// TwinCAT 3 PLC project PLC
// ProgramVersion: 3.1.4026.27
// libraries:
//   Tc2_MC2, * (Beckhoff Automation GmbH)
//   Tc2_MC2_Camming, * (Beckhoff Automation GmbH)
//   Tc2_Standard, * (Beckhoff Automation GmbH)
//   Tc2_System, * (Beckhoff Automation GmbH)
// project tree:
//   / PlcTask.TcTTO
//   DUTs/ E_Example.TcDUT, E_State.TcDUT, E_SegmentKind.TcDUT, ST_CamSegment.TcDUT, ST_CamSwitch.TcDUT
//   POUs/ F_CamPoint.TcPOU, FB_XtsBallCamBuilder.TcPOU, FB_XtsCamStitcher.TcPOU, MAIN.TcPOU, PRG_Example1.TcPOU, PRG_Example2.TcPOU, PRG_Example3.TcPOU, PRG_Example4.TcPOU, PRG_Example5.TcPOU
//   GVLs/ GVL_Axes.TcGVL
// real-time tasks:
//   TASK XTS Task 1: cycle T#250us, priority 1, ADS port 350
//   TASK XTS AUX Task 1: cycle T#250us, priority 2, ADS port 351
//   TASK PlcTask: cycle T#10ms, priority 20, ADS port 352
// motion (NC):
//   TASK NC-Task 1: cycle T#2ms, priority 4, ADS port 501
//   TASK NC-Task 1 SVB: cycle T#10ms, priority 8, ADS port 511
//   AXIS Mover Axis 1 (id 1)
//     Dynamic: AccelerationMaximum=80000, DecelerationMaximum=80000, Acceleration=20000, Deceleration=20000, Jerk=200000
//     Velo: Maximum=4000
//     PositionAreaControl: Enable=false
//     TargetPosControl: Enable=false
//     OtherSettings: AllowMotionCmdToSlave=true, AllowMotionCmdToExtSetGenAxis=true
//     encoder EncType=28
//       EncPara: ModuloFactor=1500, ToleranceWndModuloStart=0.2, MaxCount=#xffffffff
//     drive DrvType=22
//       DrvPara: MaxCount=#xffffffff, DriveControlDWord=#x00000100
//         Analog: VeloReferenz=4200, TorqueSetpointScale=10
//         TimeComp: TaskDelayCycles=1
//     controller CtrType=1
//       CtrPara: PriorControlFactor=1
//         PosDiffControl: Range=10
//         Observer: BandWidth=20
//   AXIS Mover Axis 2 (id 2)
//     Dynamic: AccelerationMaximum=80000, DecelerationMaximum=80000, Acceleration=20000, Deceleration=20000, Jerk=200000
//     Velo: Maximum=4000
//     PositionAreaControl: Enable=false
//     TargetPosControl: Enable=false
//     OtherSettings: AllowMotionCmdToSlave=true, AllowMotionCmdToExtSetGenAxis=true
//     encoder EncType=28
//       EncPara: ModuloFactor=1500, ToleranceWndModuloStart=0.2, MaxCount=#xffffffff
//     drive DrvType=22
//       DrvPara: MaxCount=#xffffffff, DriveControlDWord=#x00000100
//         Analog: VeloReferenz=4200, TorqueSetpointScale=10
//         TimeComp: TaskDelayCycles=1
//     controller CtrType=1
//       CtrPara: PriorControlFactor=1
//         PosDiffControl: Range=10
//         Observer: BandWidth=20
//   AXIS VirtualMaster (id 3)
//     General: UnitFlags=#x00000004
//     OtherSettings: AllowMotionCmdToSlave=true
//     encoder EncType=1
//       EncPara: ModuloFactor=2147.36
//     drive DrvType=5
//       Analog: TorqueSetpointScale=10, ScaleFactorActTorque=0.1
//       TimeComp: TaskDelayCycles=1
//     controller CtrType=1
//       CtrPara: PriorControlFactor=1
//         Observer: BandWidth=20
// I/O:
//   DEVICE Device 1 (disabled), AmsNetId 192.168.1.110.2.1
//     Term 0 (AT2001-0250) [AT2001-0250 Motor module with feed 250 mm, 48V]
//       Term 1 (AT2001-5250) [AT2001-5250 Sensor line with feed]
//     Term 2 (AT2050-0500) [AT2050-0500 Motor module, 90° clothoid, EtherCAT In, 48V]
//       Term 3 (AT2050-5500) [AT2050-5500 Sensor line 90° clothoid, EtherCAT In]
//     Term 4 (AT2050-0501) [AT2050-0501 Motor module, 90° clothoid, EtherCAT Out, 48V]
//       Term 5 (AT2050-5501) [AT2050-5501 Sensor line 90° clothoid, EtherCAT Out]
//     Term 6 (AT2000-0250) [AT2000-0250 Motor module 250 mm, 48V]
//       Term 7 (AT2000-5250) [AT2000-5250 Sensor line]
//     Term 8 (AT2050-0500) [AT2050-0500 Motor module, 90° clothoid, EtherCAT In, 48V]
//       Term 9 (AT2050-5500) [AT2050-5500 Sensor line 90° clothoid, EtherCAT In]
//     Term 10 (AT2050-0501) [AT2050-0501 Motor module, 90° clothoid, EtherCAT Out, 48V]
//       Term 11 (AT2050-5501) [AT2050-5501 Sensor line 90° clothoid, EtherCAT Out]
// variable links:
//   (this object) <-> TcCOM Objects/XTS ProcessingUnit 1/Part 1/Module 1
//     Term 0 (AT2001-0250)/CC Inputs/Current actual value Ch.1 <-> Data Pointer/CurrentActualValues[0]
//     Term 0 (AT2001-0250)/CC Inputs/Current actual value Ch.10 <-> Data Pointer/CurrentActualValues[9]
//     Term 0 (AT2001-0250)/CC Inputs/Current actual value Ch.11 <-> Data Pointer/CurrentActualValues[10]
//     Term 0 (AT2001-0250)/CC Inputs/Current actual value Ch.12 <-> Data Pointer/CurrentActualValues[11]
//     Term 0 (AT2001-0250)/CC Inputs/Current actual value Ch.13 <-> Data Pointer/CurrentActualValues[12]
//     Term 0 (AT2001-0250)/CC Inputs/Current actual value Ch.14 <-> Data Pointer/CurrentActualValues[13]
//     Term 0 (AT2001-0250)/CC Inputs/Current actual value Ch.15 <-> Data Pointer/CurrentActualValues[14]
//     Term 0 (AT2001-0250)/CC Inputs/Current actual value Ch.2 <-> Data Pointer/CurrentActualValues[1]
//     Term 0 (AT2001-0250)/CC Inputs/Current actual value Ch.3 <-> Data Pointer/CurrentActualValues[2]
//     Term 0 (AT2001-0250)/CC Inputs/Current actual value Ch.4 <-> Data Pointer/CurrentActualValues[3]
//     Term 0 (AT2001-0250)/CC Inputs/Current actual value Ch.5 <-> Data Pointer/CurrentActualValues[4]
//     Term 0 (AT2001-0250)/CC Inputs/Current actual value Ch.6 <-> Data Pointer/CurrentActualValues[5]
//     Term 0 (AT2001-0250)/CC Inputs/Current actual value Ch.7 <-> Data Pointer/CurrentActualValues[6]
//     Term 0 (AT2001-0250)/CC Inputs/Current actual value Ch.8 <-> Data Pointer/CurrentActualValues[7]
//     Term 0 (AT2001-0250)/CC Inputs/Current actual value Ch.9 <-> Data Pointer/CurrentActualValues[8]
//     Term 0 (AT2001-0250)/CC Inputs/Status <-> Data Pointer/Status
//     Term 0 (AT2001-0250)/CC Outputs/Control <-> Data Pointer/Control
//     Term 0 (AT2001-0250)/CC Outputs/Current setpoint value Ch.1 <-> Data Pointer/CurrentSetpointValues[0]
//     Term 0 (AT2001-0250)/CC Outputs/Current setpoint value Ch.10 <-> Data Pointer/CurrentSetpointValues[9]
//     Term 0 (AT2001-0250)/CC Outputs/Current setpoint value Ch.11 <-> Data Pointer/CurrentSetpointValues[10]
//     Term 0 (AT2001-0250)/CC Outputs/Current setpoint value Ch.12 <-> Data Pointer/CurrentSetpointValues[11]
//     Term 0 (AT2001-0250)/CC Outputs/Current setpoint value Ch.13 <-> Data Pointer/CurrentSetpointValues[12]
//     Term 0 (AT2001-0250)/CC Outputs/Current setpoint value Ch.14 <-> Data Pointer/CurrentSetpointValues[13]
//     Term 0 (AT2001-0250)/CC Outputs/Current setpoint value Ch.15 <-> Data Pointer/CurrentSetpointValues[14]
//     Term 0 (AT2001-0250)/CC Outputs/Current setpoint value Ch.2 <-> Data Pointer/CurrentSetpointValues[1]
//     Term 0 (AT2001-0250)/CC Outputs/Current setpoint value Ch.3 <-> Data Pointer/CurrentSetpointValues[2]
//     Term 0 (AT2001-0250)/CC Outputs/Current setpoint value Ch.4 <-> Data Pointer/CurrentSetpointValues[3]
//     Term 0 (AT2001-0250)/CC Outputs/Current setpoint value Ch.5 <-> Data Pointer/CurrentSetpointValues[4]
//     Term 0 (AT2001-0250)/CC Outputs/Current setpoint value Ch.6 <-> Data Pointer/CurrentSetpointValues[5]
//     Term 0 (AT2001-0250)/CC Outputs/Current setpoint value Ch.7 <-> Data Pointer/CurrentSetpointValues[6]
//     Term 0 (AT2001-0250)/CC Outputs/Current setpoint value Ch.8 <-> Data Pointer/CurrentSetpointValues[7]
//     Term 0 (AT2001-0250)/CC Outputs/Current setpoint value Ch.9 <-> Data Pointer/CurrentSetpointValues[8]
//     Term 0 (AT2001-0250)/Term 1 (AT2001-5250)/FB Inputs/Value Channel 01 <-> Data Pointer/RawPositionValues[0]
//     Term 0 (AT2001-0250)/Term 1 (AT2001-5250)/FB Inputs/Value Channel 02 <-> Data Pointer/RawPositionValues[1]
//     Term 0 (AT2001-0250)/Term 1 (AT2001-5250)/FB Inputs/Value Channel 03 <-> Data Pointer/RawPositionValues[2]
//     Term 0 (AT2001-0250)/Term 1 (AT2001-5250)/FB Inputs/Value Channel 04 <-> Data Pointer/RawPositionValues[3]
//     Term 0 (AT2001-0250)/Term 1 (AT2001-5250)/FB Inputs/Value Channel 05 <-> Data Pointer/RawPositionValues[4]
//     Term 0 (AT2001-0250)/Term 1 (AT2001-5250)/FB Inputs/Value Channel 06 <-> Data Pointer/RawPositionValues[5]
//     Term 0 (AT2001-0250)/Term 1 (AT2001-5250)/FB Inputs/Value Channel 07 <-> Data Pointer/RawPositionValues[6]
//     Term 0 (AT2001-0250)/Term 1 (AT2001-5250)/FB Inputs/Value Channel 08 <-> Data Pointer/RawPositionValues[7]
//     Term 0 (AT2001-0250)/Term 1 (AT2001-5250)/FB Inputs/Value Channel 09 <-> Data Pointer/RawPositionValues[8]
//     Term 0 (AT2001-0250)/Term 1 (AT2001-5250)/FB Inputs/Value Channel 10 <-> Data Pointer/RawPositionValues[9]
//     Term 0 (AT2001-0250)/Term 1 (AT2001-5250)/FB Inputs/Value Channel 11 <-> Data Pointer/RawPositionValues[10]
//     Term 0 (AT2001-0250)/Term 1 (AT2001-5250)/FB Inputs/Value Channel 12 <-> Data Pointer/RawPositionValues[11]
//     Term 0 (AT2001-0250)/Term 1 (AT2001-5250)/FB Inputs/Value Channel 13 <-> Data Pointer/RawPositionValues[12]
//     Term 0 (AT2001-0250)/Term 1 (AT2001-5250)/FB Inputs/Value Channel 14 <-> Data Pointer/RawPositionValues[13]
//     Term 0 (AT2001-0250)/Term 1 (AT2001-5250)/FB Inputs/Value Channel 15 <-> Data Pointer/RawPositionValues[14]
//     Term 0 (AT2001-0250)/Term 1 (AT2001-5250)/FB Inputs/Value Channel 16 <-> Data Pointer/RawPositionValues[15]
//     Term 0 (AT2001-0250)/Term 1 (AT2001-5250)/FB Inputs/Value Channel 17 <-> Data Pointer/RawPositionValues[16]
//     Term 0 (AT2001-0250)/Term 1 (AT2001-5250)/FB Inputs/Value Channel 18 <-> Data Pointer/RawPositionValues[17]
//     Term 0 (AT2001-0250)/Term 1 (AT2001-5250)/FB Inputs/Value Channel 19 <-> Data Pointer/RawPositionValues[18]
//     Term 0 (AT2001-0250)/Term 1 (AT2001-5250)/FB Inputs/Value Channel 20 <-> Data Pointer/RawPositionValues[19]
//     Term 0 (AT2001-0250)/Term 1 (AT2001-5250)/FB Inputs/Value Channel 21 <-> Data Pointer/RawPositionValues[20]
//     Term 0 (AT2001-0250)/Term 1 (AT2001-5250)/FB Inputs/Value Channel 22 <-> Data Pointer/RawPositionValues[21]
//     Term 0 (AT2001-0250)/Term 1 (AT2001-5250)/FB Inputs/Value Channel 23 <-> Data Pointer/RawPositionValues[22]
//     Term 0 (AT2001-0250)/Term 1 (AT2001-5250)/FB Inputs/Value Channel 24 <-> Data Pointer/RawPositionValues[23]
//     Term 0 (AT2001-0250)/Term 1 (AT2001-5250)/FB Inputs/Value Channel 25 <-> Data Pointer/RawPositionValues[24]
//     Term 0 (AT2001-0250)/Term 1 (AT2001-5250)/FB Inputs/Value Channel 26 <-> Data Pointer/RawPositionValues[25]
//     Term 0 (AT2001-0250)/Term 1 (AT2001-5250)/FB Inputs/Value Channel 27 <-> Data Pointer/RawPositionValues[26]
//     Term 0 (AT2001-0250)/Term 1 (AT2001-5250)/FB Inputs/Value Channel 28 <-> Data Pointer/RawPositionValues[27]
//     Term 0 (AT2001-0250)/Term 1 (AT2001-5250)/FB Inputs/Value Channel 29 <-> Data Pointer/RawPositionValues[28]
//     Term 0 (AT2001-0250)/Term 1 (AT2001-5250)/FB Inputs/Value Channel 30 <-> Data Pointer/RawPositionValues[29]
//     Term 0 (AT2001-0250)/Term 1 (AT2001-5250)/FB Inputs/Value Channel 31 <-> Data Pointer/RawPositionValues[30]
//     Term 0 (AT2001-0250)/Term 1 (AT2001-5250)/FB Inputs/Value Channel 32 <-> Data Pointer/RawPositionValues[31]
//   (this object) <-> TcCOM Objects/XTS ProcessingUnit 1/Part 1/Module 2
//     Term 2 (AT2050-0500)/CC Inputs/Current actual value Ch.1 <-> Data Pointer/CurrentActualValues[0]
//     Term 2 (AT2050-0500)/CC Inputs/Current actual value Ch.10 <-> Data Pointer/CurrentActualValues[9]
//     Term 2 (AT2050-0500)/CC Inputs/Current actual value Ch.11 <-> Data Pointer/CurrentActualValues[10]
//     Term 2 (AT2050-0500)/CC Inputs/Current actual value Ch.12 <-> Data Pointer/CurrentActualValues[11]
//     Term 2 (AT2050-0500)/CC Inputs/Current actual value Ch.13 <-> Data Pointer/CurrentActualValues[12]
//     Term 2 (AT2050-0500)/CC Inputs/Current actual value Ch.14 <-> Data Pointer/CurrentActualValues[13]
//     Term 2 (AT2050-0500)/CC Inputs/Current actual value Ch.15 <-> Data Pointer/CurrentActualValues[14]
//     Term 2 (AT2050-0500)/CC Inputs/Current actual value Ch.2 <-> Data Pointer/CurrentActualValues[1]
//     Term 2 (AT2050-0500)/CC Inputs/Current actual value Ch.3 <-> Data Pointer/CurrentActualValues[2]
//     Term 2 (AT2050-0500)/CC Inputs/Current actual value Ch.4 <-> Data Pointer/CurrentActualValues[3]
//     Term 2 (AT2050-0500)/CC Inputs/Current actual value Ch.5 <-> Data Pointer/CurrentActualValues[4]
//     Term 2 (AT2050-0500)/CC Inputs/Current actual value Ch.6 <-> Data Pointer/CurrentActualValues[5]
//     Term 2 (AT2050-0500)/CC Inputs/Current actual value Ch.7 <-> Data Pointer/CurrentActualValues[6]
//     Term 2 (AT2050-0500)/CC Inputs/Current actual value Ch.8 <-> Data Pointer/CurrentActualValues[7]
//     Term 2 (AT2050-0500)/CC Inputs/Current actual value Ch.9 <-> Data Pointer/CurrentActualValues[8]
//     Term 2 (AT2050-0500)/CC Inputs/Status <-> Data Pointer/Status
//     Term 2 (AT2050-0500)/CC Outputs/Control <-> Data Pointer/Control
//     Term 2 (AT2050-0500)/CC Outputs/Current setpoint value Ch.1 <-> Data Pointer/CurrentSetpointValues[0]
//     Term 2 (AT2050-0500)/CC Outputs/Current setpoint value Ch.10 <-> Data Pointer/CurrentSetpointValues[9]
//     Term 2 (AT2050-0500)/CC Outputs/Current setpoint value Ch.11 <-> Data Pointer/CurrentSetpointValues[10]
//     Term 2 (AT2050-0500)/CC Outputs/Current setpoint value Ch.12 <-> Data Pointer/CurrentSetpointValues[11]
//     Term 2 (AT2050-0500)/CC Outputs/Current setpoint value Ch.13 <-> Data Pointer/CurrentSetpointValues[12]
//     Term 2 (AT2050-0500)/CC Outputs/Current setpoint value Ch.14 <-> Data Pointer/CurrentSetpointValues[13]
//     Term 2 (AT2050-0500)/CC Outputs/Current setpoint value Ch.15 <-> Data Pointer/CurrentSetpointValues[14]
//     Term 2 (AT2050-0500)/CC Outputs/Current setpoint value Ch.2 <-> Data Pointer/CurrentSetpointValues[1]
//     Term 2 (AT2050-0500)/CC Outputs/Current setpoint value Ch.3 <-> Data Pointer/CurrentSetpointValues[2]
//     Term 2 (AT2050-0500)/CC Outputs/Current setpoint value Ch.4 <-> Data Pointer/CurrentSetpointValues[3]
//     Term 2 (AT2050-0500)/CC Outputs/Current setpoint value Ch.5 <-> Data Pointer/CurrentSetpointValues[4]
//     Term 2 (AT2050-0500)/CC Outputs/Current setpoint value Ch.6 <-> Data Pointer/CurrentSetpointValues[5]
//     Term 2 (AT2050-0500)/CC Outputs/Current setpoint value Ch.7 <-> Data Pointer/CurrentSetpointValues[6]
//     Term 2 (AT2050-0500)/CC Outputs/Current setpoint value Ch.8 <-> Data Pointer/CurrentSetpointValues[7]
//     Term 2 (AT2050-0500)/CC Outputs/Current setpoint value Ch.9 <-> Data Pointer/CurrentSetpointValues[8]
//     Term 2 (AT2050-0500)/Term 3 (AT2050-5500)/FB Inputs/Value Channel 01 <-> Data Pointer/RawPositionValues[0]
//     Term 2 (AT2050-0500)/Term 3 (AT2050-5500)/FB Inputs/Value Channel 02 <-> Data Pointer/RawPositionValues[1]
//     Term 2 (AT2050-0500)/Term 3 (AT2050-5500)/FB Inputs/Value Channel 03 <-> Data Pointer/RawPositionValues[2]
//     Term 2 (AT2050-0500)/Term 3 (AT2050-5500)/FB Inputs/Value Channel 04 <-> Data Pointer/RawPositionValues[3]
//     Term 2 (AT2050-0500)/Term 3 (AT2050-5500)/FB Inputs/Value Channel 05 <-> Data Pointer/RawPositionValues[4]
//     Term 2 (AT2050-0500)/Term 3 (AT2050-5500)/FB Inputs/Value Channel 06 <-> Data Pointer/RawPositionValues[5]
//     Term 2 (AT2050-0500)/Term 3 (AT2050-5500)/FB Inputs/Value Channel 07 <-> Data Pointer/RawPositionValues[6]
//     Term 2 (AT2050-0500)/Term 3 (AT2050-5500)/FB Inputs/Value Channel 08 <-> Data Pointer/RawPositionValues[7]
//     Term 2 (AT2050-0500)/Term 3 (AT2050-5500)/FB Inputs/Value Channel 09 <-> Data Pointer/RawPositionValues[8]
//     Term 2 (AT2050-0500)/Term 3 (AT2050-5500)/FB Inputs/Value Channel 10 <-> Data Pointer/RawPositionValues[9]
//     Term 2 (AT2050-0500)/Term 3 (AT2050-5500)/FB Inputs/Value Channel 11 <-> Data Pointer/RawPositionValues[10]
//     Term 2 (AT2050-0500)/Term 3 (AT2050-5500)/FB Inputs/Value Channel 12 <-> Data Pointer/RawPositionValues[11]
//     Term 2 (AT2050-0500)/Term 3 (AT2050-5500)/FB Inputs/Value Channel 13 <-> Data Pointer/RawPositionValues[12]
//     Term 2 (AT2050-0500)/Term 3 (AT2050-5500)/FB Inputs/Value Channel 14 <-> Data Pointer/RawPositionValues[13]
//     Term 2 (AT2050-0500)/Term 3 (AT2050-5500)/FB Inputs/Value Channel 15 <-> Data Pointer/RawPositionValues[14]
//     Term 2 (AT2050-0500)/Term 3 (AT2050-5500)/FB Inputs/Value Channel 16 <-> Data Pointer/RawPositionValues[15]
//     Term 2 (AT2050-0500)/Term 3 (AT2050-5500)/FB Inputs/Value Channel 17 <-> Data Pointer/RawPositionValues[16]
//     Term 2 (AT2050-0500)/Term 3 (AT2050-5500)/FB Inputs/Value Channel 18 <-> Data Pointer/RawPositionValues[17]
//     Term 2 (AT2050-0500)/Term 3 (AT2050-5500)/FB Inputs/Value Channel 19 <-> Data Pointer/RawPositionValues[18]
//     Term 2 (AT2050-0500)/Term 3 (AT2050-5500)/FB Inputs/Value Channel 20 <-> Data Pointer/RawPositionValues[19]
//     Term 2 (AT2050-0500)/Term 3 (AT2050-5500)/FB Inputs/Value Channel 21 <-> Data Pointer/RawPositionValues[20]
//     Term 2 (AT2050-0500)/Term 3 (AT2050-5500)/FB Inputs/Value Channel 22 <-> Data Pointer/RawPositionValues[21]
//     Term 2 (AT2050-0500)/Term 3 (AT2050-5500)/FB Inputs/Value Channel 23 <-> Data Pointer/RawPositionValues[22]
//     Term 2 (AT2050-0500)/Term 3 (AT2050-5500)/FB Inputs/Value Channel 24 <-> Data Pointer/RawPositionValues[23]
//     Term 2 (AT2050-0500)/Term 3 (AT2050-5500)/FB Inputs/Value Channel 25 <-> Data Pointer/RawPositionValues[24]
//     Term 2 (AT2050-0500)/Term 3 (AT2050-5500)/FB Inputs/Value Channel 26 <-> Data Pointer/RawPositionValues[25]
//     Term 2 (AT2050-0500)/Term 3 (AT2050-5500)/FB Inputs/Value Channel 27 <-> Data Pointer/RawPositionValues[26]
//     Term 2 (AT2050-0500)/Term 3 (AT2050-5500)/FB Inputs/Value Channel 28 <-> Data Pointer/RawPositionValues[27]
//     Term 2 (AT2050-0500)/Term 3 (AT2050-5500)/FB Inputs/Value Channel 29 <-> Data Pointer/RawPositionValues[28]
//     Term 2 (AT2050-0500)/Term 3 (AT2050-5500)/FB Inputs/Value Channel 30 <-> Data Pointer/RawPositionValues[29]
//     Term 2 (AT2050-0500)/Term 3 (AT2050-5500)/FB Inputs/Value Channel 31 <-> Data Pointer/RawPositionValues[30]
//     Term 2 (AT2050-0500)/Term 3 (AT2050-5500)/FB Inputs/Value Channel 32 <-> Data Pointer/RawPositionValues[31]
//   (this object) <-> TcCOM Objects/XTS ProcessingUnit 1/Part 1/Module 3
//     Term 4 (AT2050-0501)/CC Inputs/Current actual value Ch.1 <-> Data Pointer/CurrentActualValues[0]
//     Term 4 (AT2050-0501)/CC Inputs/Current actual value Ch.10 <-> Data Pointer/CurrentActualValues[9]
//     Term 4 (AT2050-0501)/CC Inputs/Current actual value Ch.11 <-> Data Pointer/CurrentActualValues[10]
//     Term 4 (AT2050-0501)/CC Inputs/Current actual value Ch.12 <-> Data Pointer/CurrentActualValues[11]
//     Term 4 (AT2050-0501)/CC Inputs/Current actual value Ch.13 <-> Data Pointer/CurrentActualValues[12]
//     Term 4 (AT2050-0501)/CC Inputs/Current actual value Ch.14 <-> Data Pointer/CurrentActualValues[13]
//     Term 4 (AT2050-0501)/CC Inputs/Current actual value Ch.15 <-> Data Pointer/CurrentActualValues[14]
//     Term 4 (AT2050-0501)/CC Inputs/Current actual value Ch.2 <-> Data Pointer/CurrentActualValues[1]
//     Term 4 (AT2050-0501)/CC Inputs/Current actual value Ch.3 <-> Data Pointer/CurrentActualValues[2]
//     Term 4 (AT2050-0501)/CC Inputs/Current actual value Ch.4 <-> Data Pointer/CurrentActualValues[3]
//     Term 4 (AT2050-0501)/CC Inputs/Current actual value Ch.5 <-> Data Pointer/CurrentActualValues[4]
//     Term 4 (AT2050-0501)/CC Inputs/Current actual value Ch.6 <-> Data Pointer/CurrentActualValues[5]
//     Term 4 (AT2050-0501)/CC Inputs/Current actual value Ch.7 <-> Data Pointer/CurrentActualValues[6]
//     Term 4 (AT2050-0501)/CC Inputs/Current actual value Ch.8 <-> Data Pointer/CurrentActualValues[7]
//     Term 4 (AT2050-0501)/CC Inputs/Current actual value Ch.9 <-> Data Pointer/CurrentActualValues[8]
//     Term 4 (AT2050-0501)/CC Inputs/Status <-> Data Pointer/Status
//     Term 4 (AT2050-0501)/CC Outputs/Control <-> Data Pointer/Control
//     Term 4 (AT2050-0501)/CC Outputs/Current setpoint value Ch.1 <-> Data Pointer/CurrentSetpointValues[0]
//     Term 4 (AT2050-0501)/CC Outputs/Current setpoint value Ch.10 <-> Data Pointer/CurrentSetpointValues[9]
//     Term 4 (AT2050-0501)/CC Outputs/Current setpoint value Ch.11 <-> Data Pointer/CurrentSetpointValues[10]
//     Term 4 (AT2050-0501)/CC Outputs/Current setpoint value Ch.12 <-> Data Pointer/CurrentSetpointValues[11]
//     Term 4 (AT2050-0501)/CC Outputs/Current setpoint value Ch.13 <-> Data Pointer/CurrentSetpointValues[12]
//     Term 4 (AT2050-0501)/CC Outputs/Current setpoint value Ch.14 <-> Data Pointer/CurrentSetpointValues[13]
//     Term 4 (AT2050-0501)/CC Outputs/Current setpoint value Ch.15 <-> Data Pointer/CurrentSetpointValues[14]
//     Term 4 (AT2050-0501)/CC Outputs/Current setpoint value Ch.2 <-> Data Pointer/CurrentSetpointValues[1]
//     Term 4 (AT2050-0501)/CC Outputs/Current setpoint value Ch.3 <-> Data Pointer/CurrentSetpointValues[2]
//     Term 4 (AT2050-0501)/CC Outputs/Current setpoint value Ch.4 <-> Data Pointer/CurrentSetpointValues[3]
//     Term 4 (AT2050-0501)/CC Outputs/Current setpoint value Ch.5 <-> Data Pointer/CurrentSetpointValues[4]
//     Term 4 (AT2050-0501)/CC Outputs/Current setpoint value Ch.6 <-> Data Pointer/CurrentSetpointValues[5]
//     Term 4 (AT2050-0501)/CC Outputs/Current setpoint value Ch.7 <-> Data Pointer/CurrentSetpointValues[6]
//     Term 4 (AT2050-0501)/CC Outputs/Current setpoint value Ch.8 <-> Data Pointer/CurrentSetpointValues[7]
//     Term 4 (AT2050-0501)/CC Outputs/Current setpoint value Ch.9 <-> Data Pointer/CurrentSetpointValues[8]
//     Term 4 (AT2050-0501)/Term 5 (AT2050-5501)/FB Inputs/Value Channel 01 <-> Data Pointer/RawPositionValues[0]
//     Term 4 (AT2050-0501)/Term 5 (AT2050-5501)/FB Inputs/Value Channel 02 <-> Data Pointer/RawPositionValues[1]
//     Term 4 (AT2050-0501)/Term 5 (AT2050-5501)/FB Inputs/Value Channel 03 <-> Data Pointer/RawPositionValues[2]
//     Term 4 (AT2050-0501)/Term 5 (AT2050-5501)/FB Inputs/Value Channel 04 <-> Data Pointer/RawPositionValues[3]
//     Term 4 (AT2050-0501)/Term 5 (AT2050-5501)/FB Inputs/Value Channel 05 <-> Data Pointer/RawPositionValues[4]
//     Term 4 (AT2050-0501)/Term 5 (AT2050-5501)/FB Inputs/Value Channel 06 <-> Data Pointer/RawPositionValues[5]
//     Term 4 (AT2050-0501)/Term 5 (AT2050-5501)/FB Inputs/Value Channel 07 <-> Data Pointer/RawPositionValues[6]
//     Term 4 (AT2050-0501)/Term 5 (AT2050-5501)/FB Inputs/Value Channel 08 <-> Data Pointer/RawPositionValues[7]
//     Term 4 (AT2050-0501)/Term 5 (AT2050-5501)/FB Inputs/Value Channel 09 <-> Data Pointer/RawPositionValues[8]
//     Term 4 (AT2050-0501)/Term 5 (AT2050-5501)/FB Inputs/Value Channel 10 <-> Data Pointer/RawPositionValues[9]
//     Term 4 (AT2050-0501)/Term 5 (AT2050-5501)/FB Inputs/Value Channel 11 <-> Data Pointer/RawPositionValues[10]
//     Term 4 (AT2050-0501)/Term 5 (AT2050-5501)/FB Inputs/Value Channel 12 <-> Data Pointer/RawPositionValues[11]
//     Term 4 (AT2050-0501)/Term 5 (AT2050-5501)/FB Inputs/Value Channel 13 <-> Data Pointer/RawPositionValues[12]
//     Term 4 (AT2050-0501)/Term 5 (AT2050-5501)/FB Inputs/Value Channel 14 <-> Data Pointer/RawPositionValues[13]
//     Term 4 (AT2050-0501)/Term 5 (AT2050-5501)/FB Inputs/Value Channel 15 <-> Data Pointer/RawPositionValues[14]
//     Term 4 (AT2050-0501)/Term 5 (AT2050-5501)/FB Inputs/Value Channel 16 <-> Data Pointer/RawPositionValues[15]
//     Term 4 (AT2050-0501)/Term 5 (AT2050-5501)/FB Inputs/Value Channel 17 <-> Data Pointer/RawPositionValues[16]
//     Term 4 (AT2050-0501)/Term 5 (AT2050-5501)/FB Inputs/Value Channel 18 <-> Data Pointer/RawPositionValues[17]
//     Term 4 (AT2050-0501)/Term 5 (AT2050-5501)/FB Inputs/Value Channel 19 <-> Data Pointer/RawPositionValues[18]
//     Term 4 (AT2050-0501)/Term 5 (AT2050-5501)/FB Inputs/Value Channel 20 <-> Data Pointer/RawPositionValues[19]
//     Term 4 (AT2050-0501)/Term 5 (AT2050-5501)/FB Inputs/Value Channel 21 <-> Data Pointer/RawPositionValues[20]
//     Term 4 (AT2050-0501)/Term 5 (AT2050-5501)/FB Inputs/Value Channel 22 <-> Data Pointer/RawPositionValues[21]
//     Term 4 (AT2050-0501)/Term 5 (AT2050-5501)/FB Inputs/Value Channel 23 <-> Data Pointer/RawPositionValues[22]
//     Term 4 (AT2050-0501)/Term 5 (AT2050-5501)/FB Inputs/Value Channel 24 <-> Data Pointer/RawPositionValues[23]
//     Term 4 (AT2050-0501)/Term 5 (AT2050-5501)/FB Inputs/Value Channel 25 <-> Data Pointer/RawPositionValues[24]
//     Term 4 (AT2050-0501)/Term 5 (AT2050-5501)/FB Inputs/Value Channel 26 <-> Data Pointer/RawPositionValues[25]
//     Term 4 (AT2050-0501)/Term 5 (AT2050-5501)/FB Inputs/Value Channel 27 <-> Data Pointer/RawPositionValues[26]
//     Term 4 (AT2050-0501)/Term 5 (AT2050-5501)/FB Inputs/Value Channel 28 <-> Data Pointer/RawPositionValues[27]
//     Term 4 (AT2050-0501)/Term 5 (AT2050-5501)/FB Inputs/Value Channel 29 <-> Data Pointer/RawPositionValues[28]
//     Term 4 (AT2050-0501)/Term 5 (AT2050-5501)/FB Inputs/Value Channel 30 <-> Data Pointer/RawPositionValues[29]
//     Term 4 (AT2050-0501)/Term 5 (AT2050-5501)/FB Inputs/Value Channel 31 <-> Data Pointer/RawPositionValues[30]
//     Term 4 (AT2050-0501)/Term 5 (AT2050-5501)/FB Inputs/Value Channel 32 <-> Data Pointer/RawPositionValues[31]
//   (this object) <-> TcCOM Objects/XTS ProcessingUnit 1/Part 1/Module 4
//     Term 6 (AT2000-0250)/CC Inputs/Current actual value Ch.1 <-> Data Pointer/CurrentActualValues[0]
//     Term 6 (AT2000-0250)/CC Inputs/Current actual value Ch.10 <-> Data Pointer/CurrentActualValues[9]
//     Term 6 (AT2000-0250)/CC Inputs/Current actual value Ch.11 <-> Data Pointer/CurrentActualValues[10]
//     Term 6 (AT2000-0250)/CC Inputs/Current actual value Ch.12 <-> Data Pointer/CurrentActualValues[11]
//     Term 6 (AT2000-0250)/CC Inputs/Current actual value Ch.13 <-> Data Pointer/CurrentActualValues[12]
//     Term 6 (AT2000-0250)/CC Inputs/Current actual value Ch.14 <-> Data Pointer/CurrentActualValues[13]
//     Term 6 (AT2000-0250)/CC Inputs/Current actual value Ch.15 <-> Data Pointer/CurrentActualValues[14]
//     Term 6 (AT2000-0250)/CC Inputs/Current actual value Ch.2 <-> Data Pointer/CurrentActualValues[1]
//     Term 6 (AT2000-0250)/CC Inputs/Current actual value Ch.3 <-> Data Pointer/CurrentActualValues[2]
//     Term 6 (AT2000-0250)/CC Inputs/Current actual value Ch.4 <-> Data Pointer/CurrentActualValues[3]
//     Term 6 (AT2000-0250)/CC Inputs/Current actual value Ch.5 <-> Data Pointer/CurrentActualValues[4]
//     Term 6 (AT2000-0250)/CC Inputs/Current actual value Ch.6 <-> Data Pointer/CurrentActualValues[5]
//     Term 6 (AT2000-0250)/CC Inputs/Current actual value Ch.7 <-> Data Pointer/CurrentActualValues[6]
//     Term 6 (AT2000-0250)/CC Inputs/Current actual value Ch.8 <-> Data Pointer/CurrentActualValues[7]
//     Term 6 (AT2000-0250)/CC Inputs/Current actual value Ch.9 <-> Data Pointer/CurrentActualValues[8]
//     Term 6 (AT2000-0250)/CC Inputs/Status <-> Data Pointer/Status
//     Term 6 (AT2000-0250)/CC Outputs/Control <-> Data Pointer/Control
//     Term 6 (AT2000-0250)/CC Outputs/Current setpoint value Ch.1 <-> Data Pointer/CurrentSetpointValues[0]
//     Term 6 (AT2000-0250)/CC Outputs/Current setpoint value Ch.10 <-> Data Pointer/CurrentSetpointValues[9]
//     Term 6 (AT2000-0250)/CC Outputs/Current setpoint value Ch.11 <-> Data Pointer/CurrentSetpointValues[10]
//     Term 6 (AT2000-0250)/CC Outputs/Current setpoint value Ch.12 <-> Data Pointer/CurrentSetpointValues[11]
//     Term 6 (AT2000-0250)/CC Outputs/Current setpoint value Ch.13 <-> Data Pointer/CurrentSetpointValues[12]
//     Term 6 (AT2000-0250)/CC Outputs/Current setpoint value Ch.14 <-> Data Pointer/CurrentSetpointValues[13]
//     Term 6 (AT2000-0250)/CC Outputs/Current setpoint value Ch.15 <-> Data Pointer/CurrentSetpointValues[14]
//     Term 6 (AT2000-0250)/CC Outputs/Current setpoint value Ch.2 <-> Data Pointer/CurrentSetpointValues[1]
//     Term 6 (AT2000-0250)/CC Outputs/Current setpoint value Ch.3 <-> Data Pointer/CurrentSetpointValues[2]
//     Term 6 (AT2000-0250)/CC Outputs/Current setpoint value Ch.4 <-> Data Pointer/CurrentSetpointValues[3]
//     Term 6 (AT2000-0250)/CC Outputs/Current setpoint value Ch.5 <-> Data Pointer/CurrentSetpointValues[4]
//     Term 6 (AT2000-0250)/CC Outputs/Current setpoint value Ch.6 <-> Data Pointer/CurrentSetpointValues[5]
//     Term 6 (AT2000-0250)/CC Outputs/Current setpoint value Ch.7 <-> Data Pointer/CurrentSetpointValues[6]
//     Term 6 (AT2000-0250)/CC Outputs/Current setpoint value Ch.8 <-> Data Pointer/CurrentSetpointValues[7]
//     Term 6 (AT2000-0250)/CC Outputs/Current setpoint value Ch.9 <-> Data Pointer/CurrentSetpointValues[8]
//     Term 6 (AT2000-0250)/Term 7 (AT2000-5250)/FB Inputs/Value Channel 01 <-> Data Pointer/RawPositionValues[0]
//     Term 6 (AT2000-0250)/Term 7 (AT2000-5250)/FB Inputs/Value Channel 02 <-> Data Pointer/RawPositionValues[1]
//     Term 6 (AT2000-0250)/Term 7 (AT2000-5250)/FB Inputs/Value Channel 03 <-> Data Pointer/RawPositionValues[2]
//     Term 6 (AT2000-0250)/Term 7 (AT2000-5250)/FB Inputs/Value Channel 04 <-> Data Pointer/RawPositionValues[3]
//     Term 6 (AT2000-0250)/Term 7 (AT2000-5250)/FB Inputs/Value Channel 05 <-> Data Pointer/RawPositionValues[4]
//     Term 6 (AT2000-0250)/Term 7 (AT2000-5250)/FB Inputs/Value Channel 06 <-> Data Pointer/RawPositionValues[5]
//     Term 6 (AT2000-0250)/Term 7 (AT2000-5250)/FB Inputs/Value Channel 07 <-> Data Pointer/RawPositionValues[6]
//     Term 6 (AT2000-0250)/Term 7 (AT2000-5250)/FB Inputs/Value Channel 08 <-> Data Pointer/RawPositionValues[7]
//     Term 6 (AT2000-0250)/Term 7 (AT2000-5250)/FB Inputs/Value Channel 09 <-> Data Pointer/RawPositionValues[8]
//     Term 6 (AT2000-0250)/Term 7 (AT2000-5250)/FB Inputs/Value Channel 10 <-> Data Pointer/RawPositionValues[9]
//     Term 6 (AT2000-0250)/Term 7 (AT2000-5250)/FB Inputs/Value Channel 11 <-> Data Pointer/RawPositionValues[10]
//     Term 6 (AT2000-0250)/Term 7 (AT2000-5250)/FB Inputs/Value Channel 12 <-> Data Pointer/RawPositionValues[11]
//     Term 6 (AT2000-0250)/Term 7 (AT2000-5250)/FB Inputs/Value Channel 13 <-> Data Pointer/RawPositionValues[12]
//     Term 6 (AT2000-0250)/Term 7 (AT2000-5250)/FB Inputs/Value Channel 14 <-> Data Pointer/RawPositionValues[13]
//     Term 6 (AT2000-0250)/Term 7 (AT2000-5250)/FB Inputs/Value Channel 15 <-> Data Pointer/RawPositionValues[14]
//     Term 6 (AT2000-0250)/Term 7 (AT2000-5250)/FB Inputs/Value Channel 16 <-> Data Pointer/RawPositionValues[15]
//     Term 6 (AT2000-0250)/Term 7 (AT2000-5250)/FB Inputs/Value Channel 17 <-> Data Pointer/RawPositionValues[16]
//     Term 6 (AT2000-0250)/Term 7 (AT2000-5250)/FB Inputs/Value Channel 18 <-> Data Pointer/RawPositionValues[17]
//     Term 6 (AT2000-0250)/Term 7 (AT2000-5250)/FB Inputs/Value Channel 19 <-> Data Pointer/RawPositionValues[18]
//     Term 6 (AT2000-0250)/Term 7 (AT2000-5250)/FB Inputs/Value Channel 20 <-> Data Pointer/RawPositionValues[19]
//     Term 6 (AT2000-0250)/Term 7 (AT2000-5250)/FB Inputs/Value Channel 21 <-> Data Pointer/RawPositionValues[20]
//     Term 6 (AT2000-0250)/Term 7 (AT2000-5250)/FB Inputs/Value Channel 22 <-> Data Pointer/RawPositionValues[21]
//     Term 6 (AT2000-0250)/Term 7 (AT2000-5250)/FB Inputs/Value Channel 23 <-> Data Pointer/RawPositionValues[22]
//     Term 6 (AT2000-0250)/Term 7 (AT2000-5250)/FB Inputs/Value Channel 24 <-> Data Pointer/RawPositionValues[23]
//     Term 6 (AT2000-0250)/Term 7 (AT2000-5250)/FB Inputs/Value Channel 25 <-> Data Pointer/RawPositionValues[24]
//     Term 6 (AT2000-0250)/Term 7 (AT2000-5250)/FB Inputs/Value Channel 26 <-> Data Pointer/RawPositionValues[25]
//     Term 6 (AT2000-0250)/Term 7 (AT2000-5250)/FB Inputs/Value Channel 27 <-> Data Pointer/RawPositionValues[26]
//     Term 6 (AT2000-0250)/Term 7 (AT2000-5250)/FB Inputs/Value Channel 28 <-> Data Pointer/RawPositionValues[27]
//     Term 6 (AT2000-0250)/Term 7 (AT2000-5250)/FB Inputs/Value Channel 29 <-> Data Pointer/RawPositionValues[28]
//     Term 6 (AT2000-0250)/Term 7 (AT2000-5250)/FB Inputs/Value Channel 30 <-> Data Pointer/RawPositionValues[29]
//     Term 6 (AT2000-0250)/Term 7 (AT2000-5250)/FB Inputs/Value Channel 31 <-> Data Pointer/RawPositionValues[30]
//     Term 6 (AT2000-0250)/Term 7 (AT2000-5250)/FB Inputs/Value Channel 32 <-> Data Pointer/RawPositionValues[31]
//   (this object) <-> TcCOM Objects/XTS ProcessingUnit 1/Part 1/Module 5
//     Term 8 (AT2050-0500)/CC Inputs/Current actual value Ch.1 <-> Data Pointer/CurrentActualValues[0]
//     Term 8 (AT2050-0500)/CC Inputs/Current actual value Ch.10 <-> Data Pointer/CurrentActualValues[9]
//     Term 8 (AT2050-0500)/CC Inputs/Current actual value Ch.11 <-> Data Pointer/CurrentActualValues[10]
//     Term 8 (AT2050-0500)/CC Inputs/Current actual value Ch.12 <-> Data Pointer/CurrentActualValues[11]
//     Term 8 (AT2050-0500)/CC Inputs/Current actual value Ch.13 <-> Data Pointer/CurrentActualValues[12]
//     Term 8 (AT2050-0500)/CC Inputs/Current actual value Ch.14 <-> Data Pointer/CurrentActualValues[13]
//     Term 8 (AT2050-0500)/CC Inputs/Current actual value Ch.15 <-> Data Pointer/CurrentActualValues[14]
//     Term 8 (AT2050-0500)/CC Inputs/Current actual value Ch.2 <-> Data Pointer/CurrentActualValues[1]
//     Term 8 (AT2050-0500)/CC Inputs/Current actual value Ch.3 <-> Data Pointer/CurrentActualValues[2]
//     Term 8 (AT2050-0500)/CC Inputs/Current actual value Ch.4 <-> Data Pointer/CurrentActualValues[3]
//     Term 8 (AT2050-0500)/CC Inputs/Current actual value Ch.5 <-> Data Pointer/CurrentActualValues[4]
//     Term 8 (AT2050-0500)/CC Inputs/Current actual value Ch.6 <-> Data Pointer/CurrentActualValues[5]
//     Term 8 (AT2050-0500)/CC Inputs/Current actual value Ch.7 <-> Data Pointer/CurrentActualValues[6]
//     Term 8 (AT2050-0500)/CC Inputs/Current actual value Ch.8 <-> Data Pointer/CurrentActualValues[7]
//     Term 8 (AT2050-0500)/CC Inputs/Current actual value Ch.9 <-> Data Pointer/CurrentActualValues[8]
//     Term 8 (AT2050-0500)/CC Inputs/Status <-> Data Pointer/Status
//     Term 8 (AT2050-0500)/CC Outputs/Control <-> Data Pointer/Control
//     Term 8 (AT2050-0500)/CC Outputs/Current setpoint value Ch.1 <-> Data Pointer/CurrentSetpointValues[0]
//     Term 8 (AT2050-0500)/CC Outputs/Current setpoint value Ch.10 <-> Data Pointer/CurrentSetpointValues[9]
//     Term 8 (AT2050-0500)/CC Outputs/Current setpoint value Ch.11 <-> Data Pointer/CurrentSetpointValues[10]
//     Term 8 (AT2050-0500)/CC Outputs/Current setpoint value Ch.12 <-> Data Pointer/CurrentSetpointValues[11]
//     Term 8 (AT2050-0500)/CC Outputs/Current setpoint value Ch.13 <-> Data Pointer/CurrentSetpointValues[12]
//     Term 8 (AT2050-0500)/CC Outputs/Current setpoint value Ch.14 <-> Data Pointer/CurrentSetpointValues[13]
//     Term 8 (AT2050-0500)/CC Outputs/Current setpoint value Ch.15 <-> Data Pointer/CurrentSetpointValues[14]
//     Term 8 (AT2050-0500)/CC Outputs/Current setpoint value Ch.2 <-> Data Pointer/CurrentSetpointValues[1]
//     Term 8 (AT2050-0500)/CC Outputs/Current setpoint value Ch.3 <-> Data Pointer/CurrentSetpointValues[2]
//     Term 8 (AT2050-0500)/CC Outputs/Current setpoint value Ch.4 <-> Data Pointer/CurrentSetpointValues[3]
//     Term 8 (AT2050-0500)/CC Outputs/Current setpoint value Ch.5 <-> Data Pointer/CurrentSetpointValues[4]
//     Term 8 (AT2050-0500)/CC Outputs/Current setpoint value Ch.6 <-> Data Pointer/CurrentSetpointValues[5]
//     Term 8 (AT2050-0500)/CC Outputs/Current setpoint value Ch.7 <-> Data Pointer/CurrentSetpointValues[6]
//     Term 8 (AT2050-0500)/CC Outputs/Current setpoint value Ch.8 <-> Data Pointer/CurrentSetpointValues[7]
//     Term 8 (AT2050-0500)/CC Outputs/Current setpoint value Ch.9 <-> Data Pointer/CurrentSetpointValues[8]
//     Term 8 (AT2050-0500)/Term 9 (AT2050-5500)/FB Inputs/Value Channel 01 <-> Data Pointer/RawPositionValues[0]
//     Term 8 (AT2050-0500)/Term 9 (AT2050-5500)/FB Inputs/Value Channel 02 <-> Data Pointer/RawPositionValues[1]
//     Term 8 (AT2050-0500)/Term 9 (AT2050-5500)/FB Inputs/Value Channel 03 <-> Data Pointer/RawPositionValues[2]
//     Term 8 (AT2050-0500)/Term 9 (AT2050-5500)/FB Inputs/Value Channel 04 <-> Data Pointer/RawPositionValues[3]
//     Term 8 (AT2050-0500)/Term 9 (AT2050-5500)/FB Inputs/Value Channel 05 <-> Data Pointer/RawPositionValues[4]
//     Term 8 (AT2050-0500)/Term 9 (AT2050-5500)/FB Inputs/Value Channel 06 <-> Data Pointer/RawPositionValues[5]
//     Term 8 (AT2050-0500)/Term 9 (AT2050-5500)/FB Inputs/Value Channel 07 <-> Data Pointer/RawPositionValues[6]
//     Term 8 (AT2050-0500)/Term 9 (AT2050-5500)/FB Inputs/Value Channel 08 <-> Data Pointer/RawPositionValues[7]
//     Term 8 (AT2050-0500)/Term 9 (AT2050-5500)/FB Inputs/Value Channel 09 <-> Data Pointer/RawPositionValues[8]
//     Term 8 (AT2050-0500)/Term 9 (AT2050-5500)/FB Inputs/Value Channel 10 <-> Data Pointer/RawPositionValues[9]
//     Term 8 (AT2050-0500)/Term 9 (AT2050-5500)/FB Inputs/Value Channel 11 <-> Data Pointer/RawPositionValues[10]
//     Term 8 (AT2050-0500)/Term 9 (AT2050-5500)/FB Inputs/Value Channel 12 <-> Data Pointer/RawPositionValues[11]
//     Term 8 (AT2050-0500)/Term 9 (AT2050-5500)/FB Inputs/Value Channel 13 <-> Data Pointer/RawPositionValues[12]
//     Term 8 (AT2050-0500)/Term 9 (AT2050-5500)/FB Inputs/Value Channel 14 <-> Data Pointer/RawPositionValues[13]
//     Term 8 (AT2050-0500)/Term 9 (AT2050-5500)/FB Inputs/Value Channel 15 <-> Data Pointer/RawPositionValues[14]
//     Term 8 (AT2050-0500)/Term 9 (AT2050-5500)/FB Inputs/Value Channel 16 <-> Data Pointer/RawPositionValues[15]
//     Term 8 (AT2050-0500)/Term 9 (AT2050-5500)/FB Inputs/Value Channel 17 <-> Data Pointer/RawPositionValues[16]
//     Term 8 (AT2050-0500)/Term 9 (AT2050-5500)/FB Inputs/Value Channel 18 <-> Data Pointer/RawPositionValues[17]
//     Term 8 (AT2050-0500)/Term 9 (AT2050-5500)/FB Inputs/Value Channel 19 <-> Data Pointer/RawPositionValues[18]
//     Term 8 (AT2050-0500)/Term 9 (AT2050-5500)/FB Inputs/Value Channel 20 <-> Data Pointer/RawPositionValues[19]
//     Term 8 (AT2050-0500)/Term 9 (AT2050-5500)/FB Inputs/Value Channel 21 <-> Data Pointer/RawPositionValues[20]
//     Term 8 (AT2050-0500)/Term 9 (AT2050-5500)/FB Inputs/Value Channel 22 <-> Data Pointer/RawPositionValues[21]
//     Term 8 (AT2050-0500)/Term 9 (AT2050-5500)/FB Inputs/Value Channel 23 <-> Data Pointer/RawPositionValues[22]
//     Term 8 (AT2050-0500)/Term 9 (AT2050-5500)/FB Inputs/Value Channel 24 <-> Data Pointer/RawPositionValues[23]
//     Term 8 (AT2050-0500)/Term 9 (AT2050-5500)/FB Inputs/Value Channel 25 <-> Data Pointer/RawPositionValues[24]
//     Term 8 (AT2050-0500)/Term 9 (AT2050-5500)/FB Inputs/Value Channel 26 <-> Data Pointer/RawPositionValues[25]
//     Term 8 (AT2050-0500)/Term 9 (AT2050-5500)/FB Inputs/Value Channel 27 <-> Data Pointer/RawPositionValues[26]
//     Term 8 (AT2050-0500)/Term 9 (AT2050-5500)/FB Inputs/Value Channel 28 <-> Data Pointer/RawPositionValues[27]
//     Term 8 (AT2050-0500)/Term 9 (AT2050-5500)/FB Inputs/Value Channel 29 <-> Data Pointer/RawPositionValues[28]
//     Term 8 (AT2050-0500)/Term 9 (AT2050-5500)/FB Inputs/Value Channel 30 <-> Data Pointer/RawPositionValues[29]
//     Term 8 (AT2050-0500)/Term 9 (AT2050-5500)/FB Inputs/Value Channel 31 <-> Data Pointer/RawPositionValues[30]
//     Term 8 (AT2050-0500)/Term 9 (AT2050-5500)/FB Inputs/Value Channel 32 <-> Data Pointer/RawPositionValues[31]
//   (this object) <-> TcCOM Objects/XTS ProcessingUnit 1/Part 1/Module 6
//     Term 10 (AT2050-0501)/CC Inputs/Current actual value Ch.1 <-> Data Pointer/CurrentActualValues[0]
//     Term 10 (AT2050-0501)/CC Inputs/Current actual value Ch.10 <-> Data Pointer/CurrentActualValues[9]
//     Term 10 (AT2050-0501)/CC Inputs/Current actual value Ch.11 <-> Data Pointer/CurrentActualValues[10]
//     Term 10 (AT2050-0501)/CC Inputs/Current actual value Ch.12 <-> Data Pointer/CurrentActualValues[11]
//     Term 10 (AT2050-0501)/CC Inputs/Current actual value Ch.13 <-> Data Pointer/CurrentActualValues[12]
//     Term 10 (AT2050-0501)/CC Inputs/Current actual value Ch.14 <-> Data Pointer/CurrentActualValues[13]
//     Term 10 (AT2050-0501)/CC Inputs/Current actual value Ch.15 <-> Data Pointer/CurrentActualValues[14]
//     Term 10 (AT2050-0501)/CC Inputs/Current actual value Ch.2 <-> Data Pointer/CurrentActualValues[1]
//     Term 10 (AT2050-0501)/CC Inputs/Current actual value Ch.3 <-> Data Pointer/CurrentActualValues[2]
//     Term 10 (AT2050-0501)/CC Inputs/Current actual value Ch.4 <-> Data Pointer/CurrentActualValues[3]
//     Term 10 (AT2050-0501)/CC Inputs/Current actual value Ch.5 <-> Data Pointer/CurrentActualValues[4]
//     Term 10 (AT2050-0501)/CC Inputs/Current actual value Ch.6 <-> Data Pointer/CurrentActualValues[5]
//     Term 10 (AT2050-0501)/CC Inputs/Current actual value Ch.7 <-> Data Pointer/CurrentActualValues[6]
//     Term 10 (AT2050-0501)/CC Inputs/Current actual value Ch.8 <-> Data Pointer/CurrentActualValues[7]
//     Term 10 (AT2050-0501)/CC Inputs/Current actual value Ch.9 <-> Data Pointer/CurrentActualValues[8]
//     Term 10 (AT2050-0501)/CC Inputs/Status <-> Data Pointer/Status
//     Term 10 (AT2050-0501)/CC Outputs/Control <-> Data Pointer/Control
//     Term 10 (AT2050-0501)/CC Outputs/Current setpoint value Ch.1 <-> Data Pointer/CurrentSetpointValues[0]
//     Term 10 (AT2050-0501)/CC Outputs/Current setpoint value Ch.10 <-> Data Pointer/CurrentSetpointValues[9]
//     Term 10 (AT2050-0501)/CC Outputs/Current setpoint value Ch.11 <-> Data Pointer/CurrentSetpointValues[10]
//     Term 10 (AT2050-0501)/CC Outputs/Current setpoint value Ch.12 <-> Data Pointer/CurrentSetpointValues[11]
//     Term 10 (AT2050-0501)/CC Outputs/Current setpoint value Ch.13 <-> Data Pointer/CurrentSetpointValues[12]
//     Term 10 (AT2050-0501)/CC Outputs/Current setpoint value Ch.14 <-> Data Pointer/CurrentSetpointValues[13]
//     Term 10 (AT2050-0501)/CC Outputs/Current setpoint value Ch.15 <-> Data Pointer/CurrentSetpointValues[14]
//     Term 10 (AT2050-0501)/CC Outputs/Current setpoint value Ch.2 <-> Data Pointer/CurrentSetpointValues[1]
//     Term 10 (AT2050-0501)/CC Outputs/Current setpoint value Ch.3 <-> Data Pointer/CurrentSetpointValues[2]
//     Term 10 (AT2050-0501)/CC Outputs/Current setpoint value Ch.4 <-> Data Pointer/CurrentSetpointValues[3]
//     Term 10 (AT2050-0501)/CC Outputs/Current setpoint value Ch.5 <-> Data Pointer/CurrentSetpointValues[4]
//     Term 10 (AT2050-0501)/CC Outputs/Current setpoint value Ch.6 <-> Data Pointer/CurrentSetpointValues[5]
//     Term 10 (AT2050-0501)/CC Outputs/Current setpoint value Ch.7 <-> Data Pointer/CurrentSetpointValues[6]
//     Term 10 (AT2050-0501)/CC Outputs/Current setpoint value Ch.8 <-> Data Pointer/CurrentSetpointValues[7]
//     Term 10 (AT2050-0501)/CC Outputs/Current setpoint value Ch.9 <-> Data Pointer/CurrentSetpointValues[8]
//     Term 10 (AT2050-0501)/Term 11 (AT2050-5501)/FB Inputs/Value Channel 01 <-> Data Pointer/RawPositionValues[0]
//     Term 10 (AT2050-0501)/Term 11 (AT2050-5501)/FB Inputs/Value Channel 02 <-> Data Pointer/RawPositionValues[1]
//     Term 10 (AT2050-0501)/Term 11 (AT2050-5501)/FB Inputs/Value Channel 03 <-> Data Pointer/RawPositionValues[2]
//     Term 10 (AT2050-0501)/Term 11 (AT2050-5501)/FB Inputs/Value Channel 04 <-> Data Pointer/RawPositionValues[3]
//     Term 10 (AT2050-0501)/Term 11 (AT2050-5501)/FB Inputs/Value Channel 05 <-> Data Pointer/RawPositionValues[4]
//     Term 10 (AT2050-0501)/Term 11 (AT2050-5501)/FB Inputs/Value Channel 06 <-> Data Pointer/RawPositionValues[5]
//     Term 10 (AT2050-0501)/Term 11 (AT2050-5501)/FB Inputs/Value Channel 07 <-> Data Pointer/RawPositionValues[6]
//     Term 10 (AT2050-0501)/Term 11 (AT2050-5501)/FB Inputs/Value Channel 08 <-> Data Pointer/RawPositionValues[7]
//     Term 10 (AT2050-0501)/Term 11 (AT2050-5501)/FB Inputs/Value Channel 09 <-> Data Pointer/RawPositionValues[8]
//     Term 10 (AT2050-0501)/Term 11 (AT2050-5501)/FB Inputs/Value Channel 10 <-> Data Pointer/RawPositionValues[9]
//     Term 10 (AT2050-0501)/Term 11 (AT2050-5501)/FB Inputs/Value Channel 11 <-> Data Pointer/RawPositionValues[10]
//     Term 10 (AT2050-0501)/Term 11 (AT2050-5501)/FB Inputs/Value Channel 12 <-> Data Pointer/RawPositionValues[11]
//     Term 10 (AT2050-0501)/Term 11 (AT2050-5501)/FB Inputs/Value Channel 13 <-> Data Pointer/RawPositionValues[12]
//     Term 10 (AT2050-0501)/Term 11 (AT2050-5501)/FB Inputs/Value Channel 14 <-> Data Pointer/RawPositionValues[13]
//     Term 10 (AT2050-0501)/Term 11 (AT2050-5501)/FB Inputs/Value Channel 15 <-> Data Pointer/RawPositionValues[14]
//     Term 10 (AT2050-0501)/Term 11 (AT2050-5501)/FB Inputs/Value Channel 16 <-> Data Pointer/RawPositionValues[15]
//     Term 10 (AT2050-0501)/Term 11 (AT2050-5501)/FB Inputs/Value Channel 17 <-> Data Pointer/RawPositionValues[16]
//     Term 10 (AT2050-0501)/Term 11 (AT2050-5501)/FB Inputs/Value Channel 18 <-> Data Pointer/RawPositionValues[17]
//     Term 10 (AT2050-0501)/Term 11 (AT2050-5501)/FB Inputs/Value Channel 19 <-> Data Pointer/RawPositionValues[18]
//     Term 10 (AT2050-0501)/Term 11 (AT2050-5501)/FB Inputs/Value Channel 20 <-> Data Pointer/RawPositionValues[19]
//     Term 10 (AT2050-0501)/Term 11 (AT2050-5501)/FB Inputs/Value Channel 21 <-> Data Pointer/RawPositionValues[20]
//     Term 10 (AT2050-0501)/Term 11 (AT2050-5501)/FB Inputs/Value Channel 22 <-> Data Pointer/RawPositionValues[21]
//     Term 10 (AT2050-0501)/Term 11 (AT2050-5501)/FB Inputs/Value Channel 23 <-> Data Pointer/RawPositionValues[22]
//     Term 10 (AT2050-0501)/Term 11 (AT2050-5501)/FB Inputs/Value Channel 24 <-> Data Pointer/RawPositionValues[23]
//     Term 10 (AT2050-0501)/Term 11 (AT2050-5501)/FB Inputs/Value Channel 25 <-> Data Pointer/RawPositionValues[24]
//     Term 10 (AT2050-0501)/Term 11 (AT2050-5501)/FB Inputs/Value Channel 26 <-> Data Pointer/RawPositionValues[25]
//     Term 10 (AT2050-0501)/Term 11 (AT2050-5501)/FB Inputs/Value Channel 27 <-> Data Pointer/RawPositionValues[26]
//     Term 10 (AT2050-0501)/Term 11 (AT2050-5501)/FB Inputs/Value Channel 28 <-> Data Pointer/RawPositionValues[27]
//     Term 10 (AT2050-0501)/Term 11 (AT2050-5501)/FB Inputs/Value Channel 29 <-> Data Pointer/RawPositionValues[28]
//     Term 10 (AT2050-0501)/Term 11 (AT2050-5501)/FB Inputs/Value Channel 30 <-> Data Pointer/RawPositionValues[29]
//     Term 10 (AT2050-0501)/Term 11 (AT2050-5501)/FB Inputs/Value Channel 31 <-> Data Pointer/RawPositionValues[30]
//     Term 10 (AT2050-0501)/Term 11 (AT2050-5501)/FB Inputs/Value Channel 32 <-> Data Pointer/RawPositionValues[31]
//   (this object) <-> NC-Task 1/Axes/Mover Axis 1
//     PlcTask Inputs/GVL_Axes.Mover1.NcToPlc <-> Outputs/ToPlc
//     PlcTask Outputs/GVL_Axes.Mover1.PlcToNc <-> Inputs/FromPlc
//   (this object) <-> NC-Task 1/Axes/Mover Axis 2
//     PlcTask Inputs/GVL_Axes.Mover2.NcToPlc <-> Outputs/ToPlc
//     PlcTask Outputs/GVL_Axes.Mover2.PlcToNc <-> Inputs/FromPlc
//   (this object) <-> NC-Task 1/Axes/VirtualMaster
//     PlcTask Inputs/GVL_Axes.VirtualMaster.NcToPlc <-> Outputs/ToPlc
//     PlcTask Outputs/GVL_Axes.VirtualMaster.PlcToNc <-> Inputs/FromPlc

CONFIGURATION PLC
    RESOURCE PLC ON TwinCAT3
        TASK PlcTask(INTERVAL := T#10ms, PRIORITY := 20);
        PROGRAM MAIN WITH PlcTask : MAIN;
    END_RESOURCE
END_CONFIGURATION

// ---- DUTs/E_Example.TcDUT
// Which example program MAIN calls. Pick one in the online view (MAIN.eExample), then start it from that program.
TYPE E_Example :
(
	ConstantGap,		// PRG_Example1: 9 points, Mover 2 a fixed distance behind Mover 1, 100 mm on the straights /
						// 60 mm in the curves (F_CamPoint)
	ClothoidBallGap,	// PRG_Example2: 18 points, the two movers pinch a ball between them like tongs and keep their
						// jaws a constant distance apart along the ball's path through the curve transitions
						// (FB_XtsBallCamBuilder)
	StitchedSegments,	// PRG_Example3: the same 18 points, assembled from a track layout and ONE module-relative
						// clothoid piece (FB_XtsCamStitcher)
	TwoTableSwitching,	// PRG_Example4: two NC tables, a 2-point straight line and the 10-point clothoid piece. The NC
						// swaps them at the curve boundaries while running
	VirtualMasterSplit	// PRG_Example5: the BALL is the master. A virtual axis runs along the ball's path at constant
						// speed and both movers follow it through their own 10-point table, so the curve work of
						// example 2 is split between them and neither ever runs faster than the ball
);
END_TYPE

// ---- DUTs/E_State.TcDUT
// Steps of the demo sequence, shared by the example programs PRG_Example1..5
TYPE E_State :
(
	Idle,			// waiting for bStart
	Enable,			// MC_Power on both movers (PRG_Example5: and on the virtual master)
	Decouple,		// MC_CamOut on a slave that is still coupled from an earlier run. The NC keeps a cam coupling through
					// an axis error and MC_Reset does not clear it; MC_CamTableSelect would then refuse the table (0x4A26)
	BuildTable,		// fill the point array(s) and load the first table into the NC (MC_CamTableSelect)
	BuildCurveTable,// PRG_Example4 only: load the clothoid piece into NC cam table 2
	LoadMover2Table,// PRG_Example5 only: load Mover 2's table into NC cam table 4 (Mover 1's went into table 3 in BuildTable)
	AlignMaster,	// PRG_Example5 only: MC_SetPosition puts the virtual master (the ball) where it belongs for Mover 1's position
	ReadTable,		// ask the NC where the table wants Mover 2 for the master's current position
	Preposition,	// move Mover 2 there (MC_MoveRelative, Mover 1 stands still)
	CamIn,			// couple the slave(s) to the master (MC_CamIn)
	Run,			// the master runs at constant velocity, the slave(s) follow the cam
	Stopping,		// MC_Halt on the master (the slaves follow it to a stop)
	CamOut,			// decouple (MC_CamOut)
	Error,			// something failed - set bReset
	Resetting		// MC_Reset on all axes
);
END_TYPE

// ---- DUTs/E_SegmentKind.TcDUT
// One piece of track as FB_XtsCamStitcher sees it (StitchedSegments example)
TYPE E_SegmentKind :
(
	Straight,	// mover path and ball path have the same length: the cam runs 1:1, no table points needed
	Curve		// one 180 deg module: the stitcher pastes the module-relative clothoid points (PRG_Example3.aCurvePoints)
);
END_TYPE

// ---- DUTs/ST_CamSegment.TcDUT
// One entry of the track layout handed to FB_XtsCamStitcher (StitchedSegments example)
TYPE ST_CamSegment :
STRUCT
	eKind	: E_SegmentKind;	// Straight or Curve
	fLength	: LREAL;			// [mm] length along the mover path (a curve module: MODULE_LENGTH, 500)
END_STRUCT
END_TYPE

// ---- DUTs/ST_CamSwitch.TcDUT
// One cam table switch of the TwoTableSwitching example: when Mover 1 passes fTrackPos, table nTableID takes over
TYPE ST_CamSwitch :
STRUCT
	fTrackPos	: LREAL;		// [mm] track position of Mover 1 (0..TRACK_LENGTH) where the NC switches
	nTableID	: MC_CAM_ID;	// cam table that becomes active there
END_STRUCT
END_TYPE

// ---- GVLs/GVL_Axes.TcGVL
// The two movers, shared by all examples (linked to NC axes "Mover Axis 1" / "Mover Axis 2").

// Only one example program runs at a time, see MAIN.
{attribute 'qualified_only'}
VAR_GLOBAL
	Mover1		  : AXIS_REF; // master
	Mover2		  : AXIS_REF; // slave
	VirtualMaster : AXIS_REF; // Virtual master
END_VAR

// ---- POUs/MAIN.TcPOU
// XTS cam table demo - as simple as it gets.
//
//   Mover 1 = master, runs at constant velocity around the track.
//   Mover 2 = slave, follows Mover 1 through a cam table.
//
// Five examples, each a self-contained program with its own constants, table builder and sequence:
//
//   PRG_Example1  ConstantGap        9 points. Mover 2 is 100 mm behind Mover 1 on the straights and 60 mm in the
//                                    curves, blended at the start of every section. Written by hand with F_CamPoint.
//   PRG_Example2  ClothoidBallGap    18 points from FB_XtsBallCamBuilder. The two movers pinch one ball between them
//                                    like tongs: each carries a jaw outboard of the track, and the table keeps the
//                                    jaws a constant distance apart along the ball's path so the ball stays clamped
//                                    through the curves (Mover 2 speeds up going in, slows down coming out).
//   PRG_Example3  StitchedSegments   The same 18 points, assembled from pieces: ONE module-relative clothoid piece
//                                    that FB_XtsCamStitcher pastes wherever the track layout says "Curve".
//   PRG_Example4  TwoTableSwitching  Two NC tables, a straight line and the clothoid piece. While running, the NC
//                                    swaps them at the curve boundaries (MC_CamIn on the coupled slave).
//   PRG_Example5  VirtualMasterSplit The BALL is the master: a virtual axis runs along the ball's path at constant
//                                    speed and BOTH movers are slaves with their own 10-point table. The curve work
//                                    that Mover 2 did alone in example 2 is split between the two movers.
//
// How to run (online view):  pick eExample here, then open that program: bStart -> watch eState -> bStop.
// On Error: bReset.   The examples share the two movers (GVL_Axes), so only the selected program is called.
// A new eExample takes effect once the running example is back in Idle.
PROGRAM MAIN
VAR
	eExample		: E_Example := E_Example.ConstantGap;	// which example to run
	eExampleActive	: E_Example;	// the one being called right now
	bIdle			: BOOL;			// the active example is in Idle, so it is safe to switch
END_VAR

CASE eExampleActive OF
	E_Example.ConstantGap:			PRG_Example1();		bIdle := PRG_Example1.eState = E_State.Idle;
	E_Example.ClothoidBallGap:		PRG_Example2();		bIdle := PRG_Example2.eState = E_State.Idle;
	E_Example.StitchedSegments:		PRG_Example3();		bIdle := PRG_Example3.eState = E_State.Idle;
	E_Example.TwoTableSwitching:	PRG_Example4();		bIdle := PRG_Example4.eState = E_State.Idle;
	E_Example.VirtualMasterSplit:	PRG_Example5();		bIdle := PRG_Example5.eState = E_State.Idle;
END_CASE

IF bIdle THEN
	eExampleActive := eExample;
END_IF

END_PROGRAM

// ---- POUs/PRG_Example1.TcPOU
// Example 1 - ConstantGap: ONE cam table, 9 points.
//
//   Mover 1 = master, runs at constant velocity around the track.
//   Mover 2 = slave, follows Mover 1 through a cam table that covers one full lap (1500 mm).
//
// Mover 2 is 100 mm behind Mover 1 on the straights and 60 mm in the curves, blended over TRANSITION mm
// at the start of every section. The table is written by hand in the action BuildTable (F_CamPoint).
//
// How to run (online view, with MAIN.eExample = ConstantGap):  bStart -> watch eState -> bStop.   On Error: bReset.
// Watch fGapActual while it runs: 100 on the straights, 60 in the curves, a smooth blend at each section start.
PROGRAM PRG_Example1
VAR CONSTANT
	// --- track geometry (mm) ---
	TRACK_LENGTH			: LREAL := 1500.0;	// = modulo factor of both mover axes
	STRAIGHT_1_START		: LREAL := 0.0;
	CURVE_1_START			: LREAL := 250.0;
	STRAIGHT_2_START		: LREAL := 750.0;
	CURVE_2_START			: LREAL := 1000.0;

	// --- wanted distance Mover 1 -> Mover 2 (mm, Mover 2 runs BEHIND Mover 1) ---
	GAP_STRAIGHT			: LREAL := 100.0;
	GAP_CURVE				: LREAL := 60.0;
	TRANSITION				: LREAL := 100.0;	// master travel over which the gap blends to the new value

	// --- demo dynamics ---
	MASTER_VELOCITY			: LREAL := 300.0;	// mm/s, Mover 1 while running
	POSITIONING_VELOCITY	: LREAL := 200.0;	// mm/s, Mover 2 while pre-positioning

	CAM_TABLE_ID			: MC_CAM_ID := 1;	// NC > Tables > Table 1 (Ex 1-4) > Mover 2
	CAM_POINTS				: UDINT := 9;
END_VAR
VAR
	// --- commands: set TRUE in the online view, they reset themselves ---
	bStart				: BOOL;
	bStop				: BOOL;
	bReset				: BOOL;
	eState				: E_State;

	// --- cam table data: CAM_POINTS points, loaded into NC table CAM_TABLE_ID ---
	aCamPoints			: ARRAY[1..CAM_POINTS] OF MC_MotionFunctionPoint;
	stCamTable			: MC_CAM_REF;

	// --- function blocks ---
	fbPowerMover1		: MC_Power;
	fbPowerMover2		: MC_Power;
	fbResetMover1		: MC_Reset;
	fbResetMover2		: MC_Reset;
	fbCamTableSelect	: MC_CamTableSelect;			// PLC array -> NC cam table
	fbReadTable			: MC_ReadCamTableSlaveDynamics;	// "where does the table want the slave for this master position?"
	fbMoveRelMover2		: MC_MoveRelative;
	fbCamIn				: MC_CamIn;
	fbMoveVeloMover1	: MC_MoveVelocity;
	fbHaltMover1		: MC_Halt;
	fbCamOut			: MC_CamOut;

	// --- live values worth watching ---
	fMover1Pos			: LREAL;	// modulo set position of Mover 1 (0..1500)
	fMover2Pos			: LREAL;	// modulo set position of Mover 2 (0..1500)
	fGapActual			: LREAL;	// how far Mover 2 is behind Mover 1 right now (along the track)
	fGapWanted			: LREAL;	// what the table asked for at coupling time
	bError				: BOOL;
	nErrorID			: UDINT;
END_VAR

// update axis status every cycle
GVL_Axes.Mover1();
GVL_Axes.Mover2();

// live gap: Mover 1 position minus Mover 2 position, wrapped to 0..1500
fMover1Pos := GVL_Axes.Mover1.NcToPlc.ModuloSetPos;
fMover2Pos := GVL_Axes.Mover2.NcToPlc.ModuloSetPos;
fGapActual := fMover1Pos - fMover2Pos;
IF fGapActual < 0.0 THEN
	fGapActual := fGapActual + TRACK_LENGTH;
END_IF

CASE eState OF
	E_State.Idle:
		IF bStart THEN
			bStart := FALSE;
			eState := E_State.Enable;
		END_IF

	E_State.Enable:
		fbPowerMover1.Enable := TRUE;
		fbPowerMover1.Enable_Positive := TRUE;
		fbPowerMover1.Enable_Negative := TRUE;
		fbPowerMover2.Enable := TRUE;
		fbPowerMover2.Enable_Positive := TRUE;
		fbPowerMover2.Enable_Negative := TRUE;
		IF fbPowerMover1.Status AND fbPowerMover2.Status THEN
			eState := E_State.Decouple;
		END_IF

	E_State.Decouple:
		// An earlier run may have left Mover 2 coupled: the NC keeps the coupling through an axis error and MC_Reset
		// does not clear it. MC_CamTableSelect refuses to overwrite a table that a coupled axis is using (0x4A26).
		IF NOT fbCamOut.Execute THEN
			IF GVL_Axes.Mover2.Status.Coupled THEN
				fbCamOut.Execute := TRUE;
			ELSE
				eState := E_State.BuildTable;
			END_IF
		ELSIF fbCamOut.Done THEN
			fbCamOut.Execute := FALSE;
			eState := E_State.BuildTable;
		END_IF

	E_State.BuildTable:
		// fill the point array once, then hand it to the NC (overwrites cam table CAM_TABLE_ID)
		IF NOT fbCamTableSelect.Execute THEN
			BuildTable();
		END_IF
		fbCamTableSelect.Periodic := TRUE;		// one table = one lap, repeat forever
		fbCamTableSelect.CamTableID := CAM_TABLE_ID;
		fbCamTableSelect.Execute := TRUE;
		IF fbCamTableSelect.Done THEN
			fbCamTableSelect.Execute := FALSE;
			eState := E_State.ReadTable;
		END_IF

	E_State.ReadTable:
		// Mover 1 stays where it is. Ask the NC what slave position the table wants for it.
		// The table master runs 0..1500 = the track, so Mover 1's track position goes in as it is.
		fbReadTable.CamTableID := CAM_TABLE_ID;
		fbReadTable.MasterPosition := fMover1Pos;
		fbReadTable.Execute := TRUE;
		IF fbReadTable.Done THEN
			fbReadTable.Execute := FALSE;
			// table: slave = master - gap   ->   gap = master - slave
			fGapWanted := fMover1Pos - fbReadTable.SlavePosition;
			// Mover 1 stands still, so this relative move can never run into it:
			// positive = Mover 2 closes up from behind, negative = Mover 2 backs off a little
			fbMoveRelMover2.Distance := fGapActual - fGapWanted;
			eState := E_State.Preposition;
		END_IF

	E_State.Preposition:
		fbMoveRelMover2.Velocity := POSITIONING_VELOCITY;
		fbMoveRelMover2.Execute := TRUE;
		IF fbMoveRelMover2.Done THEN
			fbMoveRelMover2.Execute := FALSE;
			eState := E_State.CamIn;
		END_IF

	E_State.CamIn:
		fbCamIn.CamTableID := CAM_TABLE_ID;
		fbCamIn.StartMode := MC_STARTMODE_ABSOLUTE;		// table master axis = Mover 1 track position
		fbCamIn.MasterOffset := 0.0;
		fbCamIn.SlaveOffset := 0.0;
		fbCamIn.MasterScaling := 1.0;
		fbCamIn.SlaveScaling := 1.0;
		// let the NC pick the slave offset so Mover 2 never jumps at coupling.
		// After the pre-positioning above that offset is 0 (or whole laps), so the table gaps apply 1:1.
		fbCamIn.Options.SlaveScalingMode := MC_CAMSCALING_AUTOOFFSET;
		fbCamIn.Execute := TRUE;
		IF fbCamIn.InSync THEN
			fbCamIn.Execute := FALSE;
			eState := E_State.Run;
		END_IF

	E_State.Run:
		// only the master is commanded - the slave is driven by the cam
		fbMoveVeloMover1.Velocity := MASTER_VELOCITY;
		fbMoveVeloMover1.Direction := MC_Positive_Direction;
		fbMoveVeloMover1.Execute := TRUE;
		IF bStop THEN
			bStop := FALSE;
			fbMoveVeloMover1.Execute := FALSE;
			eState := E_State.Stopping;
		END_IF

	E_State.Stopping:
		fbHaltMover1.Execute := TRUE;
		IF fbHaltMover1.Done THEN
			fbHaltMover1.Execute := FALSE;
			eState := E_State.CamOut;
		END_IF

	E_State.CamOut:
		fbCamOut.Execute := TRUE;
		IF fbCamOut.Done THEN
			fbCamOut.Execute := FALSE;
			eState := E_State.Idle;
		END_IF

	E_State.Error:
		fbCamTableSelect.Execute := FALSE;
		fbReadTable.Execute := FALSE;
		fbMoveRelMover2.Execute := FALSE;
		fbCamIn.Execute := FALSE;
		fbMoveVeloMover1.Execute := FALSE;
		// a slave error does not stop the master: halt Mover 1 if it is still running and not in error itself
		fbHaltMover1.Execute := NOT GVL_Axes.Mover1.Status.Error AND GVL_Axes.Mover1.Status.Moving;
		fbCamOut.Execute := FALSE;
		IF bReset THEN
			bReset := FALSE;
			fbResetMover1.Execute := TRUE;
			fbResetMover2.Execute := TRUE;
			eState := E_State.Resetting;
		END_IF

	E_State.Resetting:
		IF (fbResetMover1.Done OR fbResetMover1.Error) AND (fbResetMover2.Done OR fbResetMover2.Error) THEN
			fbResetMover1.Execute := FALSE;
			fbResetMover2.Execute := FALSE;
			bError := FALSE;
			nErrorID := 0;
			eState := E_State.Idle;
		END_IF
END_CASE

// any error anywhere -> Error state
IF eState <> E_State.Error AND eState <> E_State.Resetting THEN
	IF GVL_Axes.Mover1.Status.Error THEN
		nErrorID := GVL_Axes.Mover1.Status.ErrorID;
	ELSIF GVL_Axes.Mover2.Status.Error THEN
		nErrorID := GVL_Axes.Mover2.Status.ErrorID;
	ELSIF fbPowerMover1.Error THEN
		nErrorID := fbPowerMover1.ErrorID;
	ELSIF fbPowerMover2.Error THEN
		nErrorID := fbPowerMover2.ErrorID;
	ELSIF fbCamTableSelect.Error THEN
		nErrorID := fbCamTableSelect.ErrorID;
	ELSIF fbReadTable.Error THEN
		nErrorID := fbReadTable.ErrorID;
	ELSIF fbMoveRelMover2.Error THEN
		nErrorID := fbMoveRelMover2.ErrorID;
	ELSIF fbCamIn.Error THEN
		nErrorID := fbCamIn.ErrorID;
	ELSIF fbMoveVeloMover1.Error THEN
		nErrorID := fbMoveVeloMover1.ErrorID;
	ELSIF fbHaltMover1.Error THEN
		nErrorID := fbHaltMover1.ErrorID;
	ELSIF fbCamOut.Error THEN
		nErrorID := fbCamOut.ErrorID;
	END_IF
	IF nErrorID <> 0 THEN
		bError := TRUE;
		eState := E_State.Error;
	END_IF
END_IF

// call every function block once per cycle
fbPowerMover1(Axis := GVL_Axes.Mover1);
fbPowerMover2(Axis := GVL_Axes.Mover2);
fbResetMover1(Axis := GVL_Axes.Mover1);
fbResetMover2(Axis := GVL_Axes.Mover2);
fbCamTableSelect(Master := GVL_Axes.Mover1, Slave := GVL_Axes.Mover2, CamTable := stCamTable);
fbReadTable();
fbMoveRelMover2(Axis := GVL_Axes.Mover2);
fbCamIn(Master := GVL_Axes.Mover1, Slave := GVL_Axes.Mover2);
fbMoveVeloMover1(Axis := GVL_Axes.Mover1);
fbHaltMover1(Axis := GVL_Axes.Mover1);
fbCamOut(Slave := GVL_Axes.Mover2);

ACTION BuildTable:
// One lap of Mover 1 (0..1500) -> where Mover 2 has to be (master minus gap).
// Every section starts with a TRANSITION where the gap blends to the new value, then runs 1:1.
// The curve type on a point is used from that point to the NEXT point.
//
//                          idx  master position                gap           curve to next point
aCamPoints[1] := F_CamPoint(1,   STRAIGHT_1_START,              GAP_CURVE,    MOTIONFUNCTYPE_POLYNOM5_MM);	//    0: still 60 from the curve before, blend to 100
aCamPoints[2] := F_CamPoint(2,   STRAIGHT_1_START + TRANSITION, GAP_STRAIGHT, MOTIONFUNCTYPE_POLYNOM1);		//  100: 1:1, 100 behind
aCamPoints[3] := F_CamPoint(3,   CURVE_1_START,                 GAP_STRAIGHT, MOTIONFUNCTYPE_POLYNOM5_MM);	//  250: blend to 60
aCamPoints[4] := F_CamPoint(4,   CURVE_1_START + TRANSITION,    GAP_CURVE,    MOTIONFUNCTYPE_POLYNOM1);		//  350: 1:1, 60 behind
aCamPoints[5] := F_CamPoint(5,   STRAIGHT_2_START,              GAP_CURVE,    MOTIONFUNCTYPE_POLYNOM5_MM);	//  750: blend to 100
aCamPoints[6] := F_CamPoint(6,   STRAIGHT_2_START + TRANSITION, GAP_STRAIGHT, MOTIONFUNCTYPE_POLYNOM1);		//  850: 1:1, 100 behind
aCamPoints[7] := F_CamPoint(7,   CURVE_2_START,                 GAP_STRAIGHT, MOTIONFUNCTYPE_POLYNOM5_MM);	// 1000: blend to 60
aCamPoints[8] := F_CamPoint(8,   CURVE_2_START + TRANSITION,    GAP_CURVE,    MOTIONFUNCTYPE_POLYNOM1);		// 1100: 1:1, 60 behind
aCamPoints[9] := F_CamPoint(9,   TRACK_LENGTH,                  GAP_CURVE,    MOTIONFUNCTYPE_POLYNOM1);		// 1500: end of lap, same gap as point 1
aCamPoints[9].RelIndexNextPoint := 0;	// last point has no successor

// Slave goes from -60 (point 1) to 1440 (point 9) = +1500 per lap. The NC calls this a "cyclic cam
// with lift" and simply keeps adding 1500 every lap, so Mover 2 keeps going around with Mover 1.

// describe the array to the NC
stCamTable.pArray		:= ADR(aCamPoints);
stCamTable.ArraySize	:= SIZEOF(aCamPoints);
stCamTable.TableType	:= MC_TABLETYPE_MOTIONFUNCTION;
stCamTable.NoOfRows		:= CAM_POINTS;
stCamTable.NoOfColumns	:= 1;
END_ACTION

END_PROGRAM

// ---- POUs/F_CamPoint.TcPOU
// Builds one point of the motion-function cam table.
//
// Every point is a "velocity point" with slave velocity 1.0 (slave moves 1 mm per 1 mm of master)
// and acceleration 0. That is what a 1:1 relation with a fixed gap looks like.
//
// eFuncToNext is the curve type used from THIS point to the NEXT point:
//   MOTIONFUNCTYPE_POLYNOM1    - straight line   -> gap stays constant (1:1)
//   MOTIONFUNCTYPE_POLYNOM5_MM - 5th order poly  -> gap changes smoothly (motion -> motion)
//
// The slave position is written as "master minus gap", i.e. Mover 2 runs BEHIND Mover 1.
FUNCTION F_CamPoint : MC_MotionFunctionPoint
VAR_INPUT
	nIndex		: UDINT;				// 1..n, no gaps
	fMasterPos	: LREAL;				// position of Mover 1 (mm on the track)
	fGap		: LREAL;				// how far Mover 2 is behind Mover 1 at this master position (mm)
	eFuncToNext	: MC_MotionFunctionType;	// curve type towards the next point
END_VAR

F_CamPoint.PointIndex		:= nIndex;
F_CamPoint.FunctionType		:= eFuncToNext;
F_CamPoint.PointType		:= MOTIONPOINTTYPE_VELOCITY;	// velocity is given, acceleration is 0
F_CamPoint.RelIndexNextPoint	:= 1;		// next point is index+1 (the caller sets 0 on the last point)
F_CamPoint.MasterPos		:= fMasterPos;
F_CamPoint.SlavePos			:= fMasterPos - fGap;
F_CamPoint.SlaveVelo		:= 1.0;		// dSlave/dMaster = 1 -> both movers travel at the same speed here
F_CamPoint.SlaveAcc			:= 0.0;
F_CamPoint.SlaveJerk		:= 0.0;

END_FUNCTION

// ---- POUs/PRG_Example2.TcPOU
// Example 2 - ClothoidBallGap: ONE cam table, 18 points from FB_XtsBallCamBuilder.
//
//   Mover 1 = master, runs at constant velocity around the track.
//   Mover 2 = slave, follows Mover 1 through a cam table that covers one full lap (1500 mm).
//
// The two movers pinch one ball between them, like tongs: each mover carries a jaw BALL_OFFSET mm outboard of the
// track, and the table keeps the two jaws BALL_DISTANCE mm apart along the ball's path so the ball stays clamped
// through the curves. Mover 2 speeds up going into a curve and slows down coming out. The action BuildTable lets
// FB_XtsBallCamBuilder do the geometry.
//
// How to run (online view, with MAIN.eExample = ClothoidBallGap):  bStart -> watch eState -> bStop.   On Error: bReset.
// Watch fGapActual while it runs: 115 on the straights, dipping and rising through the curve transitions.
PROGRAM PRG_Example2
VAR CONSTANT
	// --- track geometry (mm) ---
	TRACK_LENGTH			: LREAL := 1500.0;	// = modulo factor of both mover axes
	CURVE_1_START			: LREAL := 250.0;
	CURVE_2_START			: LREAL := 1000.0;
	MODULE_LENGTH			: LREAL := 500.0;	// one 180 deg curve module (AT2050)

	// --- the ball clamped between the two movers ---
	BALL_DISTANCE			: LREAL := 115.0;	// mm between the two jaws, measured along the ball's path
	BALL_OFFSET				: LREAL := 103.03;	// mm the ball (and the jaws) sit outboard of the mover path
	TABLE_START				: LREAL := 180.0;	// master position of the first table point. Any point on straight 1
												// that keeps every ramp clear of the 1500 -> 0 wrap works (103 < x < 266).

	// --- demo dynamics ---
	MASTER_VELOCITY			: LREAL := 300.0;	// mm/s, Mover 1 while running
	POSITIONING_VELOCITY	: LREAL := 200.0;	// mm/s, Mover 2 while pre-positioning

	CAM_TABLE_ID			: MC_CAM_ID := 1;	// NC > Tables > Table 1 (Ex 1-4) > Mover 2
	MAX_CAM_POINTS			: UDINT := 32;		// the builder writes 8 per curve + 2 = 18, the rest is room for tuning
	PLC_ERROR_ID			: UDINT := 16#FFFF_FFFF;	// not an NC error: the builder refused, see sTableError
END_VAR
VAR
	// --- commands: set TRUE in the online view, they reset themselves ---
	bStart				: BOOL;
	bStop				: BOOL;
	bReset				: BOOL;
	eState				: E_State;

	// --- cam table data: nCamPoints points, loaded into NC table CAM_TABLE_ID ---
	aCamPoints			: ARRAY[1..MAX_CAM_POINTS] OF MC_MotionFunctionPoint;
	nCamPoints			: UDINT;		// points actually used (18)
	stCamTable			: MC_CAM_REF;
	fbBuilder			: FB_XtsBallCamBuilder;	// computes the clothoid points

	// --- function blocks ---
	fbPowerMover1		: MC_Power;
	fbPowerMover2		: MC_Power;
	fbResetMover1		: MC_Reset;
	fbResetMover2		: MC_Reset;
	fbCamTableSelect	: MC_CamTableSelect;			// PLC array -> NC cam table
	fbReadTable			: MC_ReadCamTableSlaveDynamics;	// "where does the table want the slave for this master position?"
	fbMoveRelMover2		: MC_MoveRelative;
	fbCamIn				: MC_CamIn;
	fbMoveVeloMover1	: MC_MoveVelocity;
	fbHaltMover1		: MC_Halt;
	fbCamOut			: MC_CamOut;

	// --- live values worth watching ---
	fMover1Pos			: LREAL;	// modulo set position of Mover 1 (0..1500)
	fMover2Pos			: LREAL;	// modulo set position of Mover 2 (0..1500)
	fGapActual			: LREAL;	// how far Mover 2 is behind Mover 1 right now (along the track)
	fGapWanted			: LREAL;	// what the table asked for at coupling time
	fMasterInTable		: LREAL;	// fMover1Pos mapped into the master range of the table (TABLE_START .. +1500)
	bError				: BOOL;
	nErrorID			: UDINT;
	sTableError			: STRING(255);	// why the builder refused (nErrorID = PLC_ERROR_ID)
END_VAR

// update axis status every cycle
GVL_Axes.Mover1();
GVL_Axes.Mover2();

// live gap: Mover 1 position minus Mover 2 position, wrapped to 0..1500
fMover1Pos := GVL_Axes.Mover1.NcToPlc.ModuloSetPos;
fMover2Pos := GVL_Axes.Mover2.NcToPlc.ModuloSetPos;
fGapActual := fMover1Pos - fMover2Pos;
IF fGapActual < 0.0 THEN
	fGapActual := fGapActual + TRACK_LENGTH;
END_IF

CASE eState OF
	E_State.Idle:
		IF bStart THEN
			bStart := FALSE;
			eState := E_State.Enable;
		END_IF

	E_State.Enable:
		fbPowerMover1.Enable := TRUE;
		fbPowerMover1.Enable_Positive := TRUE;
		fbPowerMover1.Enable_Negative := TRUE;
		fbPowerMover2.Enable := TRUE;
		fbPowerMover2.Enable_Positive := TRUE;
		fbPowerMover2.Enable_Negative := TRUE;
		IF fbPowerMover1.Status AND fbPowerMover2.Status THEN
			eState := E_State.Decouple;
		END_IF

	E_State.Decouple:
		// An earlier run may have left Mover 2 coupled: the NC keeps the coupling through an axis error and MC_Reset
		// does not clear it. MC_CamTableSelect refuses to overwrite a table that a coupled axis is using (0x4A26).
		IF NOT fbCamOut.Execute THEN
			IF GVL_Axes.Mover2.Status.Coupled THEN
				fbCamOut.Execute := TRUE;
			ELSE
				eState := E_State.BuildTable;
			END_IF
		ELSIF fbCamOut.Done THEN
			fbCamOut.Execute := FALSE;
			eState := E_State.BuildTable;
		END_IF

	E_State.BuildTable:
		// fill the point array once, then hand it to the NC (overwrites cam table CAM_TABLE_ID)
		IF NOT fbCamTableSelect.Execute THEN
			BuildTable();
		END_IF
		IF nCamPoints > 0 THEN		// = 0: the builder refused, the error check below picks up sTableError
			fbCamTableSelect.Periodic := TRUE;		// one table = one lap, repeat forever
			fbCamTableSelect.CamTableID := CAM_TABLE_ID;
			fbCamTableSelect.Execute := TRUE;
			IF fbCamTableSelect.Done THEN
				fbCamTableSelect.Execute := FALSE;
				eState := E_State.ReadTable;
			END_IF
		END_IF

	E_State.ReadTable:
		// Mover 1 stays where it is. Ask the NC what slave position the table wants for it.
		// The table master runs from TABLE_START to TABLE_START + 1500, so a track position
		// below the table start is one lap further on in the table.
		IF NOT fbReadTable.Execute THEN
			fMasterInTable := fMover1Pos;
			IF fMasterInTable < TABLE_START THEN
				fMasterInTable := fMasterInTable + TRACK_LENGTH;
			END_IF
			fbReadTable.CamTableID := CAM_TABLE_ID;
			fbReadTable.MasterPosition := fMasterInTable;
		END_IF
		fbReadTable.Execute := TRUE;
		IF fbReadTable.Done THEN
			fbReadTable.Execute := FALSE;
			// table: slave = master - gap   ->   gap = master - slave
			fGapWanted := fMasterInTable - fbReadTable.SlavePosition;
			// Mover 1 stands still, so this relative move can never run into it:
			// positive = Mover 2 closes up from behind, negative = Mover 2 backs off a little
			fbMoveRelMover2.Distance := fGapActual - fGapWanted;
			eState := E_State.Preposition;
		END_IF

	E_State.Preposition:
		fbMoveRelMover2.Velocity := POSITIONING_VELOCITY;
		fbMoveRelMover2.Execute := TRUE;
		IF fbMoveRelMover2.Done THEN
			fbMoveRelMover2.Execute := FALSE;
			eState := E_State.CamIn;
		END_IF

	E_State.CamIn:
		fbCamIn.CamTableID := CAM_TABLE_ID;
		fbCamIn.StartMode := MC_STARTMODE_ABSOLUTE;		// table master axis = Mover 1 track position
		fbCamIn.MasterOffset := 0.0;
		fbCamIn.SlaveOffset := 0.0;
		fbCamIn.MasterScaling := 1.0;
		fbCamIn.SlaveScaling := 1.0;
		// let the NC pick the slave offset so Mover 2 never jumps at coupling.
		// After the pre-positioning above that offset is 0 (or whole laps), so the table gaps apply 1:1.
		fbCamIn.Options.SlaveScalingMode := MC_CAMSCALING_AUTOOFFSET;
		fbCamIn.Execute := TRUE;
		IF fbCamIn.InSync THEN
			fbCamIn.Execute := FALSE;
			eState := E_State.Run;
		END_IF

	E_State.Run:
		// only the master is commanded - the slave is driven by the cam
		fbMoveVeloMover1.Velocity := MASTER_VELOCITY;
		fbMoveVeloMover1.Direction := MC_Positive_Direction;
		fbMoveVeloMover1.Execute := TRUE;
		IF bStop THEN
			bStop := FALSE;
			fbMoveVeloMover1.Execute := FALSE;
			eState := E_State.Stopping;
		END_IF

	E_State.Stopping:
		fbHaltMover1.Execute := TRUE;
		IF fbHaltMover1.Done THEN
			fbHaltMover1.Execute := FALSE;
			eState := E_State.CamOut;
		END_IF

	E_State.CamOut:
		fbCamOut.Execute := TRUE;
		IF fbCamOut.Done THEN
			fbCamOut.Execute := FALSE;
			eState := E_State.Idle;
		END_IF

	E_State.Error:
		fbCamTableSelect.Execute := FALSE;
		fbReadTable.Execute := FALSE;
		fbMoveRelMover2.Execute := FALSE;
		fbCamIn.Execute := FALSE;
		fbMoveVeloMover1.Execute := FALSE;
		// a slave error does not stop the master: halt Mover 1 if it is still running and not in error itself
		fbHaltMover1.Execute := NOT GVL_Axes.Mover1.Status.Error AND GVL_Axes.Mover1.Status.Moving;
		fbCamOut.Execute := FALSE;
		IF bReset THEN
			bReset := FALSE;
			fbResetMover1.Execute := TRUE;
			fbResetMover2.Execute := TRUE;
			eState := E_State.Resetting;
		END_IF

	E_State.Resetting:
		IF (fbResetMover1.Done OR fbResetMover1.Error) AND (fbResetMover2.Done OR fbResetMover2.Error) THEN
			fbResetMover1.Execute := FALSE;
			fbResetMover2.Execute := FALSE;
			bError := FALSE;
			nErrorID := 0;
			sTableError := '';
			eState := E_State.Idle;
		END_IF
END_CASE

// any error anywhere -> Error state
IF eState <> E_State.Error AND eState <> E_State.Resetting THEN
	IF GVL_Axes.Mover1.Status.Error THEN
		nErrorID := GVL_Axes.Mover1.Status.ErrorID;
	ELSIF GVL_Axes.Mover2.Status.Error THEN
		nErrorID := GVL_Axes.Mover2.Status.ErrorID;
	ELSIF fbPowerMover1.Error THEN
		nErrorID := fbPowerMover1.ErrorID;
	ELSIF fbPowerMover2.Error THEN
		nErrorID := fbPowerMover2.ErrorID;
	ELSIF sTableError <> '' THEN
		nErrorID := PLC_ERROR_ID;
	ELSIF fbCamTableSelect.Error THEN
		nErrorID := fbCamTableSelect.ErrorID;
	ELSIF fbReadTable.Error THEN
		nErrorID := fbReadTable.ErrorID;
	ELSIF fbMoveRelMover2.Error THEN
		nErrorID := fbMoveRelMover2.ErrorID;
	ELSIF fbCamIn.Error THEN
		nErrorID := fbCamIn.ErrorID;
	ELSIF fbMoveVeloMover1.Error THEN
		nErrorID := fbMoveVeloMover1.ErrorID;
	ELSIF fbHaltMover1.Error THEN
		nErrorID := fbHaltMover1.ErrorID;
	ELSIF fbCamOut.Error THEN
		nErrorID := fbCamOut.ErrorID;
	END_IF
	IF nErrorID <> 0 THEN
		bError := TRUE;
		eState := E_State.Error;
	END_IF
END_IF

// call every function block once per cycle
fbPowerMover1(Axis := GVL_Axes.Mover1);
fbPowerMover2(Axis := GVL_Axes.Mover2);
fbResetMover1(Axis := GVL_Axes.Mover1);
fbResetMover2(Axis := GVL_Axes.Mover2);
fbCamTableSelect(Master := GVL_Axes.Mover1, Slave := GVL_Axes.Mover2, CamTable := stCamTable);
fbReadTable();
fbMoveRelMover2(Axis := GVL_Axes.Mover2);
fbCamIn(Master := GVL_Axes.Mover1, Slave := GVL_Axes.Mover2);
fbMoveVeloMover1(Axis := GVL_Axes.Mover1);
fbHaltMover1(Axis := GVL_Axes.Mover1);
fbCamOut(Slave := GVL_Axes.Mover2);

ACTION BuildTable:
// One lap of Mover 1 (TABLE_START .. +1500) -> where Mover 2 has to be so that the two jaws stay
// BALL_DISTANCE apart along the ball's path and the ball stays clamped between them.
//
// FB_XtsBallCamBuilder does the geometry. The AT2050 curve module is not a plain half circle: its curvature
// ramps up over a short transition (a clothoid-like quintic), holds, and ramps down again. A jaw sitting
// BALL_OFFSET mm outboard of the track therefore travels further than the mover while the track is bending,
// so for the jaws to keep their distance the slave has to run faster than the master going into a curve
// and slower coming out. The builder writes 8 points per curve (ramp / plateau / ramp / line at the entry,
// mirrored at the exit) plus one point at each end of the table. See the FB header for the knot layout.
//
// Table master range 180..1680 instead of 0..1500: every ramp then lies inside the table and none of them
// straddles the 1500 -> 0 wrap of the track. The NC handles the lap mapping because the table is periodic.
sTableError := '';
nCamPoints := 0;

fbBuilder.fMasterStart		:= TABLE_START;
fbBuilder.fMasterEnd		:= TABLE_START + TRACK_LENGTH;
fbBuilder.fBallDistance		:= BALL_DISTANCE;
fbBuilder.fBallOffset		:= BALL_OFFSET;
fbBuilder.nCurves			:= 2;
fbBuilder.aCurveStart[1]	:= CURVE_1_START;
fbBuilder.aCurveStart[2]	:= CURVE_2_START;
fbBuilder.fModuleLength		:= MODULE_LENGTH;
// fTransLength, aEntryKnots, aExitKnots keep the FB defaults (tuned for 115 mm / 103 mm on AT2050 modules)
fbBuilder.pPoints			:= ADR(aCamPoints);
fbBuilder.nMaxPoints		:= MAX_CAM_POINTS;

IF NOT fbBuilder.Build() THEN
	sTableError := fbBuilder.sError;
	RETURN;
END_IF
nCamPoints := fbBuilder.nPoints;		// 18 (the builder terminates the last point itself)

// Slave goes from 65 (master 180) to 1565 (master 1680) = +1500 per lap, the same "cyclic cam with lift"
// as the ConstantGap table of example 1, so Mover 2 keeps going around with Mover 1.

// describe the array to the NC
stCamTable.pArray		:= ADR(aCamPoints);
stCamTable.ArraySize	:= nCamPoints * SIZEOF(MC_MotionFunctionPoint);
stCamTable.TableType	:= MC_TABLETYPE_MOTIONFUNCTION;
stCamTable.NoOfRows		:= nCamPoints;
stCamTable.NoOfColumns	:= 1;
END_ACTION

END_PROGRAM

// ---- POUs/FB_XtsBallCamBuilder.TcPOU
FUNCTION_BLOCK FB_XtsBallCamBuilder
(* Builds a TwinCAT motion-function cam table (MC_MotionFunctionPoint array) for two XTS movers that
   pinch one ball between them like tongs: each mover carries a jaw outward of the mover path, and the two
   jaws must keep a constant distance measured along the path of the ball so it stays clamped in the curves.
   Track: straights and 180 deg modules (Beckhoff AT2050 geometry: quintic curvature ramp + circular arc).
   Layout per module: entry ramp up (POLYNOM3) - plateau (POLYNOM1) - ramp down (POLYNOM3) - line (POLYNOM1)
                      exit  ramp down (POLYNOM3) - plateau (POLYNOM1) - ramp up (POLYNOM3) - line (POLYNOM1)
   All SlaveVelo/SlaveAcc/SlaveJerk = 0 -> TwinCAT takes the ramp end velocities from the adjacent lines.
   Generated 2026-09-16 from cam_M180-1680_D115_clothoid_xlsx_min18_p3_std.

   Second use, BuildBallMaster() (example 5): the BALL is the master. Master = distance the ball has travelled
   along its own path, slave = one mover whose jaw sits fJawLead ahead of the ball on that path. 4 points per
   module (POLYNOM5 ramp - arc line - POLYNOM5 ramp - straight line), placed exactly where that mover's jaw enters
   and leaves the curvature ramps. No tuned knots. BallArc() / InvBallArc() are public for the same reason. *)
VAR_INPUT
	// ---- cam table range ----
	fMasterStart		: LREAL := 180.0;		// [mm] master position of the first point
	fMasterEnd			: LREAL := 1680.0;		// [mm] master position of the last point
	fBallDistance		: LREAL := 115.0;		// [mm] distance master jaw -> slave jaw along the ball path (slave trails the master)

	// ---- track layout in master coordinates ----
	nCurves				: UINT  := 2;			// number of 180 deg modules inside the table range
	aCurveStart			: ARRAY[1..4] OF LREAL := [250.0, 1000.0, 0.0, 0.0];	// [mm] start of each module
	fModuleLength		: LREAL := 500.0;		// [mm] module length along the mover path (AT2050: 500)
	fTransLength		: LREAL := 84.0;		// [mm] curvature transition length at each module end (quintic ramp)
	fBallOffset			: LREAL := 103.03;		// [mm] lateral offset of the ball centre (and the jaws), outward of the mover path (r_ball - r_xts)

	// ---- knot layout, offsets relative to the module start [mm] (optimised for D = 115 mm, offset 103 mm) ----
	aEntryKnots			: ARRAY[1..4] OF LREAL := [16.0, 67.5, 90.5, 134.7];	// ramp start, plateau start, plateau end, ramp end
	aExitKnots			: ARRAY[1..4] OF LREAL := [432.0, 483.0, 493.0, 603.0];	// ramp start, plateau start, plateau end, ramp end

	// ---- options ----
	bZeroEndVelocity	: BOOL  := FALSE;		// TRUE: slave at rest at the first and last point (POLYNOM5 run-up / run-down + link line)
	fLinkLength			: LREAL := 10.0;		// [mm] POLYNOM1 link between run-up/run-down and the first/last ramp

	// ---- target buffer ----
	pPoints				: POINTER TO MC_MotionFunctionPoint;	// ADR(camPoints[first element])
	nMaxPoints			: UDINT;				// number of elements in the buffer
END_VAR
VAR_OUTPUT
	nPoints				: UDINT;				// points written (use as NoOfRows)
	fArcRadius			: LREAL;				// [mm] radius of the circular middle, derived: (fModuleLength - fTransLength) / PI
	fPeakRatio			: LREAL;				// max slave/master speed ratio = 1 + fBallOffset / fArcRadius
	bError				: BOOL;
	sError				: STRING(255);
END_VAR
VAR
	fKMax				: LREAL;				// [1/mm] curvature of the circular middle
END_VAR
VAR CONSTANT
	fPI					: LREAL := 3.14159265358979;
END_VAR

(* nothing cyclic: call Build() once *)

METHOD PRIVATE AddPoint
(* one point of the mover-master table (Build): master = leading mover, slave = trailing mover *)
VAR_INPUT
	fMaster	: LREAL;
	eFunc	: MC_MotionFunctionType;
END_VAR
AddPointXY(fMaster, SlavePos(fMaster), eFunc);
END_METHOD

METHOD PRIVATE AddPointXY
(* writes one point with an explicit slave position *)
VAR_INPUT
	fMaster	: LREAL;
	fSlave	: LREAL;
	eFunc	: MC_MotionFunctionType;
END_VAR
IF bError THEN RETURN; END_IF
IF nPoints >= nMaxPoints THEN
	bError := TRUE; sError := 'point buffer too small'; RETURN;
END_IF
IF nPoints > 0 AND_THEN fMaster <= pPoints[nPoints - 1].MasterPos THEN
	bError := TRUE; sError := CONCAT('master positions not increasing at point ', UDINT_TO_STRING(nPoints + 1)); RETURN;
END_IF

pPoints[nPoints].PointIndex        := nPoints + 1;
pPoints[nPoints].MasterPos         := fMaster;
pPoints[nPoints].SlavePos          := fSlave;
pPoints[nPoints].FunctionType      := eFunc;
pPoints[nPoints].PointType         := SEL(nPoints = 0, MC_MotionPointType.MOTIONPOINTTYPE_MOTION, MC_MotionPointType.MOTIONPOINTTYPE_ACTIVATION);
pPoints[nPoints].RelIndexNextPoint := 1;
pPoints[nPoints].SlaveVelo         := 0.0;
pPoints[nPoints].SlaveAcc          := 0.0;
pPoints[nPoints].SlaveJerk         := 0.0;
nPoints := nPoints + 1;
END_METHOD

METHOD BallArc : LREAL
(* distance the ball has travelled along its own path when the mover (its jaw) is at track position fS:
   B(s) = s + d * theta(s). Equal to s on the straight before the first module, longer after every bend. *)
VAR_INPUT
	fS	: LREAL;
END_VAR
BallArc := fS + fBallOffset * Theta(fS);
END_METHOD

METHOD Build : BOOL
VAR
	nCurve	: UINT;
	fC		: LREAL;
END_VAR
bError := FALSE; sError := ''; nPoints := 0;

IF pPoints = 0 OR nMaxPoints < 2 THEN
	bError := TRUE; sError := 'pPoints / nMaxPoints not set'; RETURN;
END_IF
IF nCurves < 1 OR nCurves > 4 THEN
	bError := TRUE; sError := 'nCurves must be 1..4'; RETURN;
END_IF
IF fTransLength <= 0 OR fTransLength >= 0.5 * fModuleLength THEN
	bError := TRUE; sError := 'fTransLength out of range'; RETURN;
END_IF

// 180 deg over the module: kmax * (L_mod - L_trans) = PI  (the quintic ramp integrates to half its length)
fKMax      := fPI / (fModuleLength - fTransLength);
fArcRadius := 1.0 / fKMax;
fPeakRatio := 1.0 + fBallOffset * fKMax;

// ---- first point(s) ----
IF bZeroEndVelocity THEN
	AddPoint(fMasterStart, MC_MotionFunctionType.MOTIONFUNCTYPE_POLYNOM5);								// run-up from rest
	AddPoint(aCurveStart[1] + aEntryKnots[1] - fLinkLength, MC_MotionFunctionType.MOTIONFUNCTYPE_POLYNOM1);	// short line
ELSE
	AddPoint(fMasterStart, MC_MotionFunctionType.MOTIONFUNCTYPE_POLYNOM1);
END_IF

// ---- per module: entry (ratio 1 -> peak -> 1) and exit (ratio 1 -> 1/peak -> 1) ----
FOR nCurve := 1 TO nCurves DO
	fC := aCurveStart[nCurve];
	AddPoint(fC + aEntryKnots[1], MC_MotionFunctionType.MOTIONFUNCTYPE_POLYNOM3);	// ramp up
	AddPoint(fC + aEntryKnots[2], MC_MotionFunctionType.MOTIONFUNCTYPE_POLYNOM1);	// plateau at the ratio maximum
	AddPoint(fC + aEntryKnots[3], MC_MotionFunctionType.MOTIONFUNCTYPE_POLYNOM3);	// ramp down
	AddPoint(fC + aEntryKnots[4], MC_MotionFunctionType.MOTIONFUNCTYPE_POLYNOM1);	// both on the arc: ratio 1
	AddPoint(fC + aExitKnots[1],  MC_MotionFunctionType.MOTIONFUNCTYPE_POLYNOM3);	// ramp down
	AddPoint(fC + aExitKnots[2],  MC_MotionFunctionType.MOTIONFUNCTYPE_POLYNOM1);	// plateau at the ratio minimum
	AddPoint(fC + aExitKnots[3],  MC_MotionFunctionType.MOTIONFUNCTYPE_POLYNOM3);	// ramp up
	AddPoint(fC + aExitKnots[4],  MC_MotionFunctionType.MOTIONFUNCTYPE_POLYNOM1);	// both on the straight: ratio 1
END_FOR

// ---- last point(s) ----
IF bZeroEndVelocity THEN
	AddPoint(aCurveStart[nCurves] + aExitKnots[4] + fLinkLength, MC_MotionFunctionType.MOTIONFUNCTYPE_POLYNOM5);	// run-down to rest
END_IF
AddPoint(fMasterEnd, MC_MotionFunctionType.MOTIONFUNCTYPE_POLYNOM1);

IF NOT bError THEN
	pPoints[nPoints - 1].RelIndexNextPoint := 0;	// terminate the table
END_IF
Build := NOT bError;
END_METHOD

METHOD BuildBallMaster : BOOL
(* Cam table for a master that is the BALL, for ONE of the two movers (call it twice, once per mover).
   Master = distance the ball has travelled along its own path [mm]. The table covers one lap of the track,
            BallArc(fMasterStart) .. BallArc(fMasterEnd); its period is the track length + 2 pi * fBallOffset.
   Slave  = track position of the mover whose jaw sits fJawLead mm AHEAD of the ball along the ball's path:
            +fBallDistance/2 for the leading mover, -fBallDistance/2 for the trailing one.
   On a straight the mover runs at the ball's speed (ratio 1). While its jaw is in an arc the ball travels further
   than the mover, so the mover runs at 1/fPeakRatio. The change happens exactly while the jaw is in a curvature
   ramp of the module, so the knots are the ramp ends and need no tuning: 4 points per module + 2.
   Ramps are POLYNOM5 between two lines: position and velocity from the lines, acceleration 0 at both ends,
   as in the true profile. Both movers get the same curve, shifted by fBallDistance along the master. *)
VAR_INPUT
	fJawLead	: LREAL;		// [mm] jaw position ahead of the ball along the ball's path (negative = behind)
END_VAR
VAR
	nCurve	: UINT;
	fC		: LREAL;
END_VAR
bError := FALSE; sError := ''; nPoints := 0;

IF pPoints = 0 OR nMaxPoints < 2 THEN
	bError := TRUE; sError := 'pPoints / nMaxPoints not set'; RETURN;
END_IF
IF nCurves < 1 OR nCurves > 4 THEN
	bError := TRUE; sError := 'nCurves must be 1..4'; RETURN;
END_IF
IF fTransLength <= 0 OR fTransLength >= 0.5 * fModuleLength THEN
	bError := TRUE; sError := 'fTransLength out of range'; RETURN;
END_IF

fKMax      := fPI / (fModuleLength - fTransLength);
fArcRadius := 1.0 / fKMax;
fPeakRatio := 1.0 + fBallOffset * fKMax;

// ---- first point: on the straight, ratio 1 ----
AddBallPoint(BallArc(fMasterStart), fJawLead, MC_MotionFunctionType.MOTIONFUNCTYPE_POLYNOM1);

// ---- per module: the jaw enters the ramp (slow down), rides the arc, enters the exit ramp (speed up), is out ----
FOR nCurve := 1 TO nCurves DO
	fC := aCurveStart[nCurve];
	AddBallPoint(BallArc(fC) - fJawLead,                             fJawLead, MC_MotionFunctionType.MOTIONFUNCTYPE_POLYNOM5);	// ratio 1 -> 1/peak
	AddBallPoint(BallArc(fC + fTransLength) - fJawLead,              fJawLead, MC_MotionFunctionType.MOTIONFUNCTYPE_POLYNOM1);	// on the arc: 1/peak
	AddBallPoint(BallArc(fC + fModuleLength - fTransLength) - fJawLead, fJawLead, MC_MotionFunctionType.MOTIONFUNCTYPE_POLYNOM5);	// 1/peak -> 1
	AddBallPoint(BallArc(fC + fModuleLength) - fJawLead,             fJawLead, MC_MotionFunctionType.MOTIONFUNCTYPE_POLYNOM1);	// on the straight: 1
END_FOR

// ---- last point ----
AddBallPoint(BallArc(fMasterEnd), fJawLead, MC_MotionFunctionType.MOTIONFUNCTYPE_POLYNOM1);

IF NOT bError THEN
	pPoints[nPoints - 1].RelIndexNextPoint := 0;	// terminate the table
END_IF
BuildBallMaster := NOT bError;
END_METHOD

METHOD PRIVATE AddBallPoint
(* one point of a ball-master table (BuildBallMaster): master = ball path position, slave = the mover whose jaw
   is fJawLead ahead of the ball on that path *)
VAR_INPUT
	fBallPos	: LREAL;
	fJawLead	: LREAL;
	eFunc		: MC_MotionFunctionType;
END_VAR
AddPointXY(fBallPos, InvBallArc(fBallPos + fJawLead), eFunc);
END_METHOD

METHOD InvBallArc : LREAL
(* the inverse of BallArc: mover (jaw) track position for a ball path length. Newton iteration on B(s) = fB *)
VAR_INPUT
	fB	: LREAL;
END_VAR
VAR
	fS, fF	: LREAL;
	i		: UINT;
END_VAR
fS := fB;
FOR i := 1 TO 50 DO
	fF := BallArc(fS) - fB;
	IF ABS(fF) < 1.0E-9 THEN EXIT; END_IF
	fS := fS - fF / (1.0 + fBallOffset * Kappa(fS));
END_FOR
InvBallArc := fS;
END_METHOD

METHOD PRIVATE Kappa : LREAL
(* curvature [1/mm] of the mover path at fS *)
VAR_INPUT
	fS	: LREAL;
END_VAR
VAR
	i	: UINT;
END_VAR
Kappa := 0.0;
FOR i := 1 TO nCurves DO
	Kappa := Kappa + KappaMod(fS - aCurveStart[i]);
END_FOR
END_METHOD

METHOD PRIVATE KappaMod : LREAL
(* curvature inside one 180 deg module, fU = position from module start.
   Quintic ramp k = kmax * (10 t^3 - 15 t^4 + 6 t^5), t = u / L_trans; circular middle; mirrored ramp *)
VAR_INPUT
	fU	: LREAL;
END_VAR
VAR
	t	: LREAL;
END_VAR
IF fU <= 0.0 OR fU >= fModuleLength THEN
	KappaMod := 0.0;
ELSIF fU < fTransLength THEN
	t := fU / fTransLength;
	KappaMod := fKMax * t * t * t * (10.0 - 15.0 * t + 6.0 * t * t);
ELSIF fU <= fModuleLength - fTransLength THEN
	KappaMod := fKMax;
ELSE
	t := (fModuleLength - fU) / fTransLength;
	KappaMod := fKMax * t * t * t * (10.0 - 15.0 * t + 6.0 * t * t);
END_IF
END_METHOD

METHOD SlavePos : LREAL
(* exact slave position for a master position: constant distance fBallDistance along the ball path *)
VAR_INPUT
	fMaster	: LREAL;
END_VAR
SlavePos := InvBallArc(BallArc(fMaster) - fBallDistance);
END_METHOD

METHOD SpeedRatio : LREAL
(* exact slave/master speed ratio ds/dm for a master position (diagnostics) *)
VAR_INPUT
	fMaster	: LREAL;
END_VAR
SpeedRatio := (1.0 + fBallOffset * Kappa(fMaster)) / (1.0 + fBallOffset * Kappa(SlavePos(fMaster)));
END_METHOD

METHOD PRIVATE Theta : LREAL
(* heading angle [rad] turned between fMasterStart and fS (sum over the modules; table covers one lap) *)
VAR_INPUT
	fS	: LREAL;
END_VAR
VAR
	i	: UINT;
END_VAR
Theta := 0.0;
FOR i := 1 TO nCurves DO
	Theta := Theta + ThetaMod(fS - aCurveStart[i]);
END_FOR
END_METHOD

METHOD PRIVATE ThetaMod : LREAL
(* heading [rad] turned inside one module up to fU (closed-form integral of KappaMod):
   ramp: kmax * L_trans * (2.5 t^4 - 3 t^5 + t^6); a full ramp turns kmax * L_trans / 2 *)
VAR_INPUT
	fU	: LREAL;
END_VAR
VAR
	t	: LREAL;
END_VAR
IF fU <= 0.0 THEN
	ThetaMod := 0.0;
ELSIF fU >= fModuleLength THEN
	ThetaMod := fPI;
ELSIF fU < fTransLength THEN
	t := fU / fTransLength;
	ThetaMod := fKMax * fTransLength * t * t * t * t * (2.5 - 3.0 * t + t * t);
ELSIF fU <= fModuleLength - fTransLength THEN
	ThetaMod := 0.5 * fKMax * fTransLength + fKMax * (fU - fTransLength);
ELSE
	t := (fModuleLength - fU) / fTransLength;
	ThetaMod := fPI - fKMax * fTransLength * t * t * t * t * (2.5 - 3.0 * t + t * t);
END_IF
END_METHOD

END_FUNCTION_BLOCK

// ---- POUs/PRG_Example3.TcPOU
// Example 3 - StitchedSegments: ONE cam table, the same 18 points as example 2, assembled from pieces.
//
//   Mover 1 = master, runs at constant velocity around the track.
//   Mover 2 = slave, follows Mover 1 through a cam table that covers one full lap (1500 mm).
//
// The clothoid exists once, as a module-relative piece: BuildCurveModule runs FB_XtsBallCamBuilder for ONE curve
// module at the origin (aCurvePoints). The track is a list of segments, and FB_XtsCamStitcher pastes the piece
// wherever the list says "Curve" (action BuildTable). Change the straights = change the list, the clothoid stays.
//
// How to run (online view, with MAIN.eExample = StitchedSegments):  bStart -> watch eState -> bStop.   On Error: bReset.
// Watch fGapActual while it runs (115 on the straights) and fStitchMaxDeviation: the difference to the example 2
// table, expect ~1e-9 mm.
PROGRAM PRG_Example3
VAR CONSTANT
	// --- track geometry (mm) ---
	TRACK_LENGTH			: LREAL := 1500.0;	// = modulo factor of both mover axes
	STRAIGHT_1_START		: LREAL := 0.0;
	CURVE_1_START			: LREAL := 250.0;
	STRAIGHT_2_START		: LREAL := 750.0;
	CURVE_2_START			: LREAL := 1000.0;
	MODULE_LENGTH			: LREAL := 500.0;	// one 180 deg curve module (AT2050)

	// --- the ball clamped between the two movers (see example 2) ---
	BALL_DISTANCE			: LREAL := 115.0;	// mm between the two jaws, measured along the ball's path
	BALL_OFFSET				: LREAL := 103.03;	// mm the ball (and the jaws) sit outboard of the mover path
	TABLE_START				: LREAL := 180.0;	// master position of the first table point. Any point on straight 1
												// that keeps every ramp clear of the 1500 -> 0 wrap works (103 < x < 266).

	// --- the clothoid as ONE module-relative piece ---
	CURVE_TABLE_LENGTH		: LREAL := 620.0;	// mm of master one curve piece covers, measured from the module start.
												// Must reach past the builder's last exit knot (603): the trailing ball
												// keeps the cam busy 103 mm after the module ends. The builder errors if not.
	MAX_CURVE_POINTS		: UDINT := 16;

	// --- demo dynamics ---
	MASTER_VELOCITY			: LREAL := 300.0;	// mm/s, Mover 1 while running
	POSITIONING_VELOCITY	: LREAL := 200.0;	// mm/s, Mover 2 while pre-positioning

	CAM_TABLE_ID			: MC_CAM_ID := 1;	// NC > Tables > Table 1 (Ex 1-4) > Mover 2
	MAX_CAM_POINTS			: UDINT := 32;		// 8 per curve + 2 = 18, the rest is room for more segments
	PLC_ERROR_ID			: UDINT := 16#FFFF_FFFF;	// not an NC error: builder or stitcher refused, see sTableError
END_VAR
VAR
	// --- commands: set TRUE in the online view, they reset themselves ---
	bStart				: BOOL;
	bStop				: BOOL;
	bReset				: BOOL;
	eState				: E_State;

	// --- cam table data: nCamPoints points, loaded into NC table CAM_TABLE_ID ---
	aCamPoints			: ARRAY[1..MAX_CAM_POINTS] OF MC_MotionFunctionPoint;
	nCamPoints			: UDINT;		// points actually used (18)
	stCamTable			: MC_CAM_REF;

	// --- the clothoid piece and the stitcher ---
	fbBuilder			: FB_XtsBallCamBuilder;	// computes the clothoid points of one module
	aCurvePoints		: ARRAY[1..MAX_CURVE_POINTS] OF MC_MotionFunctionPoint;	// 10 points, master 0..CURVE_TABLE_LENGTH from the module start
	nCurvePoints		: UDINT;
	fbStitcher			: FB_XtsCamStitcher;	// layout + curve piece -> one lap table
	aCheckPoints		: ARRAY[1..MAX_CAM_POINTS] OF MC_MotionFunctionPoint;	// the example 2 table, built next to it for comparison
	fStitchMaxDeviation	: LREAL;		// largest difference to the example 2 table in mm (expect ~1e-9, -1 = no comparison)

	// --- function blocks ---
	fbPowerMover1		: MC_Power;
	fbPowerMover2		: MC_Power;
	fbResetMover1		: MC_Reset;
	fbResetMover2		: MC_Reset;
	fbCamTableSelect	: MC_CamTableSelect;			// PLC array -> NC cam table
	fbReadTable			: MC_ReadCamTableSlaveDynamics;	// "where does the table want the slave for this master position?"
	fbMoveRelMover2		: MC_MoveRelative;
	fbCamIn				: MC_CamIn;
	fbMoveVeloMover1	: MC_MoveVelocity;
	fbHaltMover1		: MC_Halt;
	fbCamOut			: MC_CamOut;

	// --- live values worth watching ---
	fMover1Pos			: LREAL;	// modulo set position of Mover 1 (0..1500)
	fMover2Pos			: LREAL;	// modulo set position of Mover 2 (0..1500)
	fGapActual			: LREAL;	// how far Mover 2 is behind Mover 1 right now (along the track)
	fGapWanted			: LREAL;	// what the table asked for at coupling time
	fMasterInTable		: LREAL;	// fMover1Pos mapped into the master range of the table (TABLE_START .. +1500)
	bError				: BOOL;
	nErrorID			: UDINT;
	sTableError			: STRING(255);	// why the PLC side refused: builder or stitcher (nErrorID = PLC_ERROR_ID)

	// --- scratch ---
	i					: UINT;
END_VAR

// update axis status every cycle
GVL_Axes.Mover1();
GVL_Axes.Mover2();

// live gap: Mover 1 position minus Mover 2 position, wrapped to 0..1500
fMover1Pos := GVL_Axes.Mover1.NcToPlc.ModuloSetPos;
fMover2Pos := GVL_Axes.Mover2.NcToPlc.ModuloSetPos;
fGapActual := fMover1Pos - fMover2Pos;
IF fGapActual < 0.0 THEN
	fGapActual := fGapActual + TRACK_LENGTH;
END_IF

CASE eState OF
	E_State.Idle:
		IF bStart THEN
			bStart := FALSE;
			eState := E_State.Enable;
		END_IF

	E_State.Enable:
		fbPowerMover1.Enable := TRUE;
		fbPowerMover1.Enable_Positive := TRUE;
		fbPowerMover1.Enable_Negative := TRUE;
		fbPowerMover2.Enable := TRUE;
		fbPowerMover2.Enable_Positive := TRUE;
		fbPowerMover2.Enable_Negative := TRUE;
		IF fbPowerMover1.Status AND fbPowerMover2.Status THEN
			eState := E_State.Decouple;
		END_IF

	E_State.Decouple:
		// An earlier run may have left Mover 2 coupled: the NC keeps the coupling through an axis error and MC_Reset
		// does not clear it. MC_CamTableSelect refuses to overwrite a table that a coupled axis is using (0x4A26).
		IF NOT fbCamOut.Execute THEN
			IF GVL_Axes.Mover2.Status.Coupled THEN
				fbCamOut.Execute := TRUE;
			ELSE
				eState := E_State.BuildTable;
			END_IF
		ELSIF fbCamOut.Done THEN
			fbCamOut.Execute := FALSE;
			eState := E_State.BuildTable;
		END_IF

	E_State.BuildTable:
		// fill the point array once, then hand it to the NC (overwrites cam table CAM_TABLE_ID)
		IF NOT fbCamTableSelect.Execute THEN
			BuildTable();
		END_IF
		IF nCamPoints > 0 THEN		// = 0: builder or stitcher refused, the error check below picks up sTableError
			fbCamTableSelect.Periodic := TRUE;		// one table = one lap, repeat forever
			fbCamTableSelect.CamTableID := CAM_TABLE_ID;
			fbCamTableSelect.Execute := TRUE;
			IF fbCamTableSelect.Done THEN
				fbCamTableSelect.Execute := FALSE;
				eState := E_State.ReadTable;
			END_IF
		END_IF

